(* CODESYS project ChiefMaster.project

Project tree, tasks and I/O mapping:
  Device : HY-TTC 580, TTControl, order no. n/a, version 1.7.1.0
    application Application
      libraries: Standard, * (System); lib500_can2, 0.2.0.5 (TTControl); lib500, 1.7.1.0 (TTControl); lib500_types, 1.7.1.0 (TTControl); lib500_syscom, 1.7.1.0 (TTControl)
      task MainTask (cyclic, interval t#10ms, priority 2, watchdog t#30ms x 1) calls PLC_PRG
      program PLC_PRG [ST]
      global variables GVL
      function block Receive [ST]
      function block Transmit [ST]
      function block Chart [ST]
      global variables GVL_CONSTS
      global variables GVL_VARS
      function block PLC_CODER_TIMER [ST]
      function rt_floorf [ST]
      function block Lib_InputProcessing_state [ST]
      function rt_floord [ST]
      function block Chart1 [ST]
      function block Chart1_l [ST]
      function block Chart_ContactorFB_State_Batt1 [ST]
      function block Chart_lg [ST]
      function block ChiefMaster [ST]
      function block Chart_REQ_IMD_ON_BB1 [ST]
      function block Chart_REQ_IMD_ON_BB2 [ST]
      function block Chart_REQ_IMD_ON_BB3 [ST]
      function block Chart_WeldingDetection [ST]
      function block Chart_j [ST]
      function block VoltageDetermination [ST]
      function PLC_BOOL_TO_LREAL [ST]
      function block InsulationMonitoringReq [ST]
      function block Chart_ek [ST]
      function block Chart_ls [ST]
      function block fcn_EmergencyButtonState [ST]
      function block Chart_REQ_HV_ON_Batt1 [ST]
      function block BattChargeFcn [ST]
      function block Chart_PrechargeStatus [ST]
      function block Chart_REQ_MAIN_MINUS [ST]
      function block SafeToCloseHV [ST]
      function block HVIL_NOK [ST]
      function block Chart_SetDominantSwitch [ST]
      function block Chart_ContactorFB_State_Batt2 [ST]
      function block Chart_ContactorFB_State_Batt3 [ST]
      function block CMState [ST]
      function block EmergencySD [ST]
      function block IMD_SD [ST]
      function block SDError [ST]
      function block Chart_Hysteresis_LowActive [ST]
      function block BDU_Error [ST]
      function block ChartBatt1 [ST]
      function block Chartbatt2 [ST]
      function block ChartBatt3 [ST]
      function block Input_Delay [ST]
      function block Chart_REQ_HV_ON_Batt2 [ST]
      function block Chart_REQ_HV_ON_Batt3 [ST]
      function block REQ_HV_ON_Batt [ST]
      function block Chart_Hysteresis_HighActive [ST]
      function block HVIL_Input_Delay [ST]
      function block IMDOK_Input_Delay [ST]
      function block EMSRET [ST]
      function block EMSRET_Power [ST]
      function block Chart_jj [ST]
      function block Chart_m [ST]
      function block IMD_OK [ST]
      function IMD_Error [ST]
    CANs : CANs, TTControl, order no. n/a, version 1.7.1.0
      CAN0 : CAN0, TTControl, order no. n/a, version 1.7.1.0
      CAN1 : CAN1, TTControl, order no. n/a, version 1.7.1.0
      CAN2 : CAN2, TTControl, order no. n/a, version 1.7.1.0
          settings: Baudrate = 250
      CAN3 : CAN3, TTControl, order no. n/a, version 1.7.1.0
      CAN4 : CAN4, TTControl, order no. n/a, version 1.7.1.0
          settings: Baudrate = 250
      CAN5 : CAN5, TTControl, order no. n/a, version 1.7.1.0
          settings: Baudrate = 250
      CAN6 : CAN6, TTControl, order no. n/a, version 1.7.1.0
    System : System, TTControl, order no. n/a, version 1.7.1.0
        output Application.GVL.gPowerStage : BYTE  // mode
        output Application.GVL.gSafetySwitch0 : BYTE  // mode
        output Application.GVL.gSafetySwitch1 : BYTE  // mode
        output Application.GVL.gSafetySwitch2 : BYTE  // mode
        output Application.GVL.gSensorSupply0 : BYTE  // mode
        output Application.GVL.gSensorSupply1 : BYTE  // mode
        output Application.GVL.gSensorSupply2 : BYTE  // mode
        output TTC_Sleep : BIT  // shutdown
        input  VBat_mV : DWORD  // UBAT.value
        input  KL15_mV : DWORD  // Terminal_15.value
        input  WakeUp_mV : DWORD  // WakeUp.value
        input  WakeUp : BYTE  // WakeUp.state
        unmapped channels: error, error, error, error, error, error, error, error, enable_error_group_0, enable_error_group_1, enable_error_group_2, diag_status, safe_state, error, driver_init_error, UBAT, Terminal_15, WakeUp, Temperature, SSW0, SSW1, SSW2, SSUP0, SSUP1, SSUP2, status, write, boot_error, trigger_error, Powerstage, SSW0, SSW1, SSW2, SSUP0, SSUP1, SSUP2, Terminal_15, WakeUp, ExtShutOff0, ExtShutOff1,
          ExtShutOff2
      Analog_Inputs_2Mode_10V : AIN_2Mode_10V, TTControl, order no. n/a, version 1.7.1.0
        Pin 107
          HVIL_BDU : IoDrvADC2Mode10, TTControl, order no. n/a, version 1.7.1.0
              input  AI_HVIL_BDU_P107 : DWORD  // status.value
              unmapped channels: status, reset_trigger, reset_count, reset_error
        Pin 131
          EmergencyButton_NC : IoDrvADC2Mode10, TTControl, order no. n/a, version 1.7.1.0
              input  AI_EmergencyButton_NC_P131 : DWORD  // status.value
              unmapped channels: status, reset_trigger, reset_count, reset_error
        Pin 108
          HVIL_Components : IoDrvADC2Mode10, TTControl, order no. n/a, version 1.7.1.0
              input  AI_HVIL_Components_P108 : DWORD  // status.value
              unmapped channels: status, reset_trigger, reset_count, reset_error
        Pin 132
          ResetButton_NO : IoDrvDILim, TTControl, order no. n/a, version 1.7.1.0
              input  DI_ResetButton_NO_P132 : BIT  // status.pin_value
              unmapped channels: status
        Pin 109
          HVIL_Battery : IoDrvADC2Mode10, TTControl, order no. n/a, version 1.7.1.0
              input  AI_HVIL_Battery_P109 : DWORD  // status.value
              unmapped channels: status, reset_trigger, reset_count, reset_error
        Pin 133
          Proximity_BB1 : IoDrvDILim, TTControl, order no. n/a, version 1.7.1.0
              input  DI_Proximity_BB1_P133 : BIT  // status.pin_value
              unmapped channels: status
        Pin 110
          HVIL_Overrule : IoDrvDILim, TTControl, order no. n/a, version 1.7.1.0
              input  DI_HVIL_Overrule_P110 : BIT  // status.pin_value
              unmapped channels: status
        Pin 134
          Proximity_BB2 : IoDrvDILim, TTControl, order no. n/a, version 1.7.1.0
              input  DI_Proximity_BB2_P134 : BIT  // status.pin_value
              unmapped channels: status
      Analog_Inputs_2Mode_32V : AIN_2Mode_32V, TTControl, order no. n/a, version 1.7.1.0
        Pin 111
          <Empty>
        Pin 135
          Proximity_BB3 : IoDrvDILim, TTControl, order no. n/a, version 1.7.1.0
              input  DI_Proximity_BB3_P135 : BIT  // status.pin_value
              unmapped channels: status
        Pin 112
          IMD_FB_BB1 : IoDrvDILim, TTControl, order no. n/a, version 1.7.1.0
              input  DI_IMD_FB_BB1_P112 : BIT  // status.pin_value
              unmapped channels: status
        Pin 136
          <Empty>
        Pin 113
          IMD_FB_BB2 : IoDrvDILim, TTControl, order no. n/a, version 1.7.1.0
              input  DI_IMD_FB_BB2_P113 : BIT  // status.pin_value
              unmapped channels: status
        Pin 137
          <Empty>
        Pin 114
          IMD_FB_BB3 : IoDrvDILim, TTControl, order no. n/a, version 1.7.1.0
              input  DI_IMD_FB_BB3_P114 : BIT  // status.pin_value
              unmapped channels: status
        Pin 138
          <Empty>
      Analog_Inputs_3Mode : AIN_3Mode, TTControl, order no. n/a, version 1.7.1.0
        Pin 103
          <Empty>
        Pin 127
          <Empty>
        Pin 104
          <Empty>
        Pin 128
          <Empty>
        Pin 105
          <Empty>
        Pin 129
          <Empty>
        Pin 106
          <Empty>
        Pin 130
          <Empty>
      Digital_Outputs_HS : HSDOUT, TTControl, order no. n/a, version 1.7.1.0
        Pin 149
          KL15_BB1 : IoDrvDOSafety, TTControl, order no. n/a, version 1.7.1.0
              output DO_KL15_BB1_P149 : BIT  // output
              unmapped channels: error_code, reset_trigger, reset_count, reset_error, current, voltage_feedback
        Pin 173
          IMD_BB1 : IoDrvDOSafety, TTControl, order no. n/a, version 1.7.1.0
              output DO_IMD_BB1_P173 : BIT  // output
              unmapped channels: error_code, reset_trigger, reset_count, reset_error, current, voltage_feedback
        Pin 152
          KL15_BB2 : IoDrvDOSafety, TTControl, order no. n/a, version 1.7.1.0
              output DO_KL15_BB2_P152 : BIT  // output
              unmapped channels: error_code, reset_trigger, reset_count, reset_error, current, voltage_feedback
        Pin 176
          IMD_BB2 : IoDrvDOSafety, TTControl, order no. n/a, version 1.7.1.0
              output DO_IMD_BB2_P176 : BIT  // output
              unmapped channels: error_code, reset_trigger, reset_count, reset_error, current, voltage_feedback
        Pin 155
          KL15_BB3 : IoDrvDOSafety, TTControl, order no. n/a, version 1.7.1.0
              output DO_KL15_BB3_P155 : BIT  // output
              unmapped channels: error_code, reset_trigger, reset_count, reset_error, current, voltage_feedback
        Pin 179
          IMD_BB3 : IoDrvDOSafety, TTControl, order no. n/a, version 1.7.1.0
              output DO_IMD_BB3_P179 : BIT  // output
              unmapped channels: error_code, reset_trigger, reset_count, reset_error, current, voltage_feedback
        Pin 158
          <Empty>
        Pin 182
          <Empty>
      Digital_Outputs_LS : LSDOUT, TTControl, order no. n/a, version 1.7.1.0
        Pin 251
          Request_Main_Precharge : IoDrvDO, TTControl, order no. n/a, version 1.7.1.0
              output DO_Request_Main_Precharge_P251 : BIT  // output
              unmapped channels: error_code, reset_trigger, reset_count, reset_error, current
        Pin 238
          Request_Main_Plus : IoDrvDO, TTControl, order no. n/a, version 1.7.1.0
              output DO_Request_Main_Plus_P238 : BIT  // output
              unmapped channels: error_code, reset_trigger, reset_count, reset_error, current
        Pin 252
          <Empty>
        Pin 239
          Request_Main_Minus : IoDrvDO, TTControl, order no. n/a, version 1.7.1.0
              output DO_Request_Main_Minus_P239 : BIT  // output
              unmapped channels: error_code, reset_trigger, reset_count, reset_error, current
        Pin 253
          <Empty>
        Pin 240
          Request_DC_Plus : IoDrvDO, TTControl, order no. n/a, version 1.7.1.0
              output DO_Request_DC_Plus_P240 : BIT  // output
              unmapped channels: error_code, reset_trigger, reset_count, reset_error, current
        Pin 254
          <Empty>
        Pin 241
          Request_DC_Minus : IoDrvDO, TTControl, order no. n/a, version 1.7.1.0
              output DO_Request_DC_Minus_P241 : BIT  // output
              unmapped channels: error_code, reset_trigger, reset_count, reset_error, current
      PVG_Outputs : PVG, TTControl, order no. n/a, version 1.7.1.0
        Pin 161
          HVIL_Supply : IoDrvDODiag, TTControl, order no. n/a, version 1.7.1.0
              settings: diagnostic = FALSE
              output DO_HVIL_Supply_P161 : BIT  // output
              unmapped channels: error_code, reset_trigger, reset_count, reset_error, current, voltage_feedback
        Pin 185
          ResetButton_LED : IoDrvDODiag, TTControl, order no. n/a, version 1.7.1.0
              settings: diagnostic = FALSE
              output DO_REsetButton_LED_P185 : BIT  // output
              unmapped channels: error_code, reset_trigger, reset_count, reset_error, current, voltage_feedback
        Pin 188
          CabinAlarm : IoDrvDODiag, TTControl, order no. n/a, version 1.7.1.0
              settings: diagnostic = FALSE
              output DO_CabinAlarm_P188 : BIT  // output
              unmapped channels: error_code, reset_trigger, reset_count, reset_error, current, voltage_feedback
        Pin 164
          <Empty>
        Pin 191
          <Empty>
        Pin 167
          <Empty>
        Pin 194
          <Empty>
        Pin 170
          <Empty>
      PWM_Outputs : PWM, TTControl, order no. n/a, version 1.7.1.0
        Safety_switch_0 : PWM_SSW0, TTControl, order no. n/a, version 1.7.1.0
          Pin 153
            <Empty>
          Pin 177
            HeaterPump : IoDrvDO, TTControl, order no. n/a, version 1.7.1.0
                output DO_HeaterPump_Active_Pin177 : BIT  // output
                unmapped channels: error_code, reset_trigger, reset_count, reset_error, current
          Pin 156
            <Empty>
          Pin 180
            Alternator_ouput : IoDrvDO, TTControl, order no. n/a, version 1.7.1.0
                output DO_AlternatorOutput_Pin180 : BIT  // output
                unmapped channels: error_code, reset_trigger, reset_count, reset_error, current
          Pin 159
            <Empty>
          Pin 183
            CoolingSystemPump : IoDrvDO, TTControl, order no. n/a, version 1.7.1.0
                output DO_CoolingSystemPump_Pin183 : BIT  // output
                unmapped channels: error_code, reset_trigger, reset_count, reset_error, current
          Pin 186
            CoolingSystemFan : IoDrvDO, TTControl, order no. n/a, version 1.7.1.0
                output DO_CoolingSystemFan_Pin186 : BIT  // output
                unmapped channels: error_code, reset_trigger, reset_count, reset_error, current
          Pin 162
            <Empty>
          Pin 189
            HydraulicFan : IoDrvDO, TTControl, order no. n/a, version 1.7.1.0
                output DO_HydraulicFan_Pin189 : BIT  // output
                unmapped channels: error_code, reset_trigger, reset_count, reset_error, current
          Pin 165
            <Empty>
          Pin 192
            BMS_KL15 : IoDrvDO, TTControl, order no. n/a, version 1.7.1.0
                output DO_BMSKL15_Pin192 : BIT  // output
                unmapped channels: error_code, reset_trigger, reset_count, reset_error, current
          Pin 168
            <Empty>
          Pin 195
            <Empty>
          Pin 171
            <Empty>
        Safety_switch_1 : PWM_SSW1, TTControl, order no. n/a, version 1.7.1.0
          Pin 154
            <Empty>
          Pin 178
            <Empty>
          Pin 157
            <Empty>
          Pin 181
            <Empty>
          Pin 160
            <Empty>
          Pin 184
            <Empty>
          Pin 187
            <Empty>
          Pin 163
            <Empty>
          Pin 190
            <Empty>
          Pin 166
            <Empty>
          Pin 193
            <Empty>
          Pin 169
            <Empty>
          Pin 196
            <Empty>
          Pin 172
            <Empty>
        Safety_switch_2 : PWM_SSW2, TTControl, order no. n/a, version 1.7.1.0
          Pin 101
            EMSRET_BDU1 : IoDrvDO, TTControl, order no. n/a, version 1.7.1.0
                output DO_EMSRET_BDU1 : BIT  // output
                unmapped channels: error_code, reset_trigger, reset_count, reset_error, current
          Pin 125
            EMSRET_BDU2 : IoDrvDO, TTControl, order no. n/a, version 1.7.1.0
                output DO_EMSRET_BDU2 : BIT  // output
                unmapped channels: error_code, reset_trigger, reset_count, reset_error, current
          Pin 150
            EMSRET_BB2_1 : IoDrvDO, TTControl, order no. n/a, version 1.7.1.0
                output DO_EMSRET_BB2_1 : BIT  // output
                unmapped channels: error_code, reset_trigger, reset_count, reset_error, current
          Pin 174
            EMSRET_BB2_2 : IoDrvDO, TTControl, order no. n/a, version 1.7.1.0
                output DO_EMSRET_BB2_2 : BIT  // output
                unmapped channels: error_code, reset_trigger, reset_count, reset_error, current
          Pin 102
            EMSRET_BB1_1 : IoDrvDO, TTControl, order no. n/a, version 1.7.1.0
                output DO_EMSRET_BB1_1 : BIT  // output
                unmapped channels: error_code, reset_trigger, reset_count, reset_error, current
          Pin 126
            EMSRET_BB1_2 : IoDrvDO, TTControl, order no. n/a, version 1.7.1.0
                output DO_EMSRET_BB1_2 : BIT  // output
                unmapped channels: error_code, reset_trigger, reset_count, reset_error, current
          Pin 151
            EMSRET_BB3_1 : IoDrvDO, TTControl, order no. n/a, version 1.7.1.0
                output DO_EMSRET_BB3_1 : BIT  // output
                unmapped channels: error_code, reset_trigger, reset_count, reset_error, current
          Pin 175
            EMSRET_BB3_2 : IoDrvDO, TTControl, order no. n/a, version 1.7.1.0
                output DO_EMSRET_BB3_2 : BIT  // output
                unmapped channels: error_code, reset_trigger, reset_count, reset_error, current
      Timer_Inputs_Cur : TIN_Cur, TTControl, order no. n/a, version 1.7.1.0
        Pin 115
          Main_Plus_FB : IoDrvADC, TTControl, order no. n/a, version 1.7.1.0
              input  AI_Main_Plus_FB_P115 : DWORD  // status.value
              unmapped channels: status
        Pin 139
          <Empty>
        Pin 116
          Main_Minus_FB : IoDrvADC, TTControl, order no. n/a, version 1.7.1.0
              input  AI_Main_Minus_FB_P116 : DWORD  // status.value
              unmapped channels: status
        Pin 140
          <Empty>
        Pin 117
          <Empty>
        Pin 141
          <Empty>
      Timer_Inputs : TIN, TTControl, order no. n/a, version 1.7.1.0
        Pin 122
          DC_Plus_FB : IoDrvADC, TTControl, order no. n/a, version 1.7.1.0
              input  AI_DC_Plus_FB_P122 : DWORD  // status.value
              unmapped channels: status
        Pin 146
          <Empty>
        Pin 123
          DC_Minus_FB : IoDrvADC, TTControl, order no. n/a, version 1.7.1.0
              input  AI_DC_Minus_FB_P123 : DWORD  // status.value
              unmapped channels: status
        Pin 147
          <Empty>
        Pin 124
          <Empty>
        Pin 148
          <Empty>
*)

// Device/Application/GVL
 {attribute 'qualified_only'}
VAR_GLOBAL
	(*System*)
	gPowerStage    : lib500_types.IO_POWER_STATE := lib500_types.IO_POWER_STATE.IO_POWER_OFF;	(* Powerstage status variable *)
	gSafetySwitch0 : lib500_types.IO_POWER_STATE := lib500_types.IO_POWER_STATE.IO_POWER_OFF;   (* Safey Switch 0 status variable *)
	gSafetySwitch1 : lib500_types.IO_POWER_STATE := lib500_types.IO_POWER_STATE.IO_POWER_OFF;   (* Safey Switch 1 status variable *)
	gSafetySwitch2 : lib500_types.IO_POWER_STATE := lib500_types.IO_POWER_STATE.IO_POWER_OFF;   (* Safey Switch 2 status variable *)
	gSensorSupply0 : lib500_types.IO_POWER_STATE := lib500_types.IO_POWER_STATE.IO_POWER_OFF;   (* Sensor Supply status variable *)
	gSensorSupply1 : lib500_types.IO_POWER_STATE := lib500_types.IO_POWER_STATE.IO_POWER_OFF;   (* Sensor Supply status variable *)
	gSensorSupply2 : lib500_types.IO_POWER_STATE := lib500_types.IO_POWER_STATE.IO_POWER_OFF;   (* Sensor Supply status variable *)
	G_tonCMSleep_timer:TON;
	G_CMSleep: BOOL;
	
(*CAN*)
	gCan0: tCan;
	gCan1: tCan;
	gCan2: tCan;
	gCan3: tCan;
	gCan4: tCan;
	gCan5: tCan;

	(*Recieve*)
	
(*Actia*)
(*Box 1*)
	C_Actia_BB1_MyStatus: ARRAY [0..7] OF BYTE;
	C_Actia_BB1_MyStatus_Timeout: BOOL;
	C_Actia_BB1_Error: ARRAY [0..7] OF BYTE;
	C_Actia_BB1_Error_Timeout: BOOL;
	C_Actia_BB1_ADS_8: ARRAY [0..7] OF BYTE;
	C_Actia_BB1_ADS_8_Timeout: BOOL;
	C_Actia_BB1_ADS_0: ARRAY [0..7] OF BYTE;
	C_Actia_BB1_ADS_0_Timeout: BOOL;
	C_Actia_BB1_ADS_1: ARRAY [0..7] OF BYTE;
	C_Actia_BB1_ADS_1_Timeout: BOOL;
	C_Actia_BB1_ADS_3: ARRAY [0..7] OF BYTE;
	C_Actia_BB1_ADS_3_Timeout: BOOL;
(*Box 2*)
	C_Actia_BB2_MyStatus: ARRAY [0..7] OF BYTE;
	C_Actia_BB2_MyStatus_Timeout: BOOL;
	C_Actia_BB2_Error: ARRAY [0..7] OF BYTE;
	C_Actia_BB2_Error_Timeout: BOOL;
	C_Actia_BB2_ADS_8: ARRAY [0..7] OF BYTE;
	C_Actia_BB2_ADS_8_Timeout: BOOL;
	C_Actia_BB2_ADS_0: ARRAY [0..7] OF BYTE;
	C_Actia_BB2_ADS_0_Timeout: BOOL;
	C_Actia_BB2_ADS_1: ARRAY [0..7] OF BYTE;
	C_Actia_BB2_ADS_1_Timeout: BOOL;
	C_Actia_BB2_ADS_3: ARRAY [0..7] OF BYTE;
	C_Actia_BB2_ADS_3_Timeout: BOOL;
(*Box 3*)	
	C_Actia_BB3_MyStatus: ARRAY [0..7] OF BYTE;
	C_Actia_BB3_MyStatus_Timeout: BOOL;
	C_Actia_BB3_Error: ARRAY [0..7] OF BYTE;
	C_Actia_BB3_Error_Timeout: BOOL;
	C_Actia_BB3_ADS_8: ARRAY [0..7] OF BYTE;
	C_Actia_BB3_ADS_8_Timeout: BOOL;
	C_Actia_BB3_ADS_0: ARRAY [0..7] OF BYTE;
	C_Actia_BB3_ADS_0_Timeout: BOOL;
	C_Actia_BB3_ADS_1: ARRAY [0..7] OF BYTE;
	C_Actia_BB3_ADS_1_Timeout: BOOL;
	C_Actia_BB3_ADS_3: ARRAY [0..7] OF BYTE;
	C_Actia_BB3_ADS_3_Timeout: BOOL;
	
(*LiBa*)
(*Box 1*)
	C_LB_Batt1_CellVoltage01: ARRAY[0..7] OF BYTE;
	C_LB_Batt1_CellVoltage01_Timeout: BOOL;
	C_LB_Batt1_CellVoltage02: ARRAY[0..7] OF BYTE;
	C_LB_Batt1_CellVoltage02_Timeout: BOOL;
	C_LB_Batt1_CellTemperature: ARRAY[0..7] OF BYTE;
	C_LB_Batt1_CellTemperature_Timeout: BOOL;
	C_LB_Batt1_InsulationMonitor: ARRAY[0..7] OF BYTE;
	C_LB_Batt1_InsulationMonitor_Timeout: BOOL;
	C_LB_Batt1_Status01: ARRAY[0..7] OF BYTE;
	C_LB_Batt1_Status01_Timeout: BOOL;
	C_LB_Batt1_Status02: ARRAY[0..7] OF BYTE;
	C_LB_Batt1_Status02_Timeout: BOOL;
	C_LB_Batt1_Status03: ARRAY[0..7] OF BYTE;
	C_LB_Batt1_Status03_Timeout: BOOL;

(*Box 2*)
	C_LB_Batt2_CellVoltage01: ARRAY[0..7] OF BYTE;
	C_LB_Batt2_CellVoltage01_Timeout: BOOL;
	C_LB_Batt2_CellVoltage02: ARRAY[0..7] OF BYTE;
	C_LB_Batt2_CellVoltage02_Timeout: BOOL;
	C_LB_Batt2_CellTemperature: ARRAY[0..7] OF BYTE;
	C_LB_Batt2_CellTemperature_Timeout: BOOL;
	C_LB_Batt2_InsulationMonitor: ARRAY[0..7] OF BYTE;
	C_LB_Batt2_InsulationMonitor_Timeout: BOOL;
	C_LB_Batt2_Status01: ARRAY[0..7] OF BYTE;
	C_LB_Batt2_Status01_Timeout: BOOL;
	C_LB_Batt2_Status02: ARRAY[0..7] OF BYTE;
	C_LB_Batt2_Status02_Timeout: BOOL;
	C_LB_Batt2_Status03: ARRAY[0..7] OF BYTE;
	C_LB_Batt2_Status03_Timeout: BOOL;

(*Box 3*)
	C_LB_Batt3_CellVoltage01: ARRAY[0..7] OF BYTE;
	C_LB_Batt3_CellVoltage01_Timeout: BOOL;
	C_LB_Batt3_CellVoltage02: ARRAY[0..7] OF BYTE;
	C_LB_Batt3_CellVoltage02_Timeout: BOOL;
	C_LB_Batt3_CellTemperature: ARRAY[0..7] OF BYTE;
	C_LB_Batt3_CellTemperature_Timeout: BOOL;
	C_LB_Batt3_InsulationMonitor: ARRAY[0..7] OF BYTE;
	C_LB_Batt3_InsulationMonitor_Timeout: BOOL;
	C_LB_Batt3_Status01: ARRAY[0..7] OF BYTE;
	C_LB_Batt3_Status01_Timeout: BOOL;
	C_LB_Batt3_Status02: ARRAY[0..7] OF BYTE;
	C_LB_Batt3_Status02_Timeout: BOOL;
	C_LB_Batt3_Status03: ARRAY[0..7] OF BYTE;
	C_LB_Batt3_Status03_Timeout: BOOL;
	
(*UDC*)	
	C_UDC_Msg1: ARRAY[0..7] OF BYTE;
	C_UDC_Msg1_Timeout: BOOL;
	
(*Transmit*)
(*Actia*)
	C_Actia_Control_Batt1 : ARRAY[0..7] OF BYTE;
	C_Actia_Control_Batt2 : ARRAY[0..7] OF BYTE;
	C_Actia_Control_Batt3 : ARRAY[0..7] OF BYTE;
(*LiBa*)
	C_LiBa_OperationRequest_Batt1: ARRAY[0..7] OF BYTE;
	C_LiBa_OperationRequest_Batt2: ARRAY[0..7] OF BYTE;
	C_LiBa_OperationRequest_Batt3: ARRAY[0..7] OF BYTE;
(*Chief Master*)
	C_Chief_Master_Msg1 : ARRAY[0..7] OF BYTE;
	C_Chief_Master_Msg2 : ARRAY[0..7] OF BYTE;
	C_Chief_Master_Msg3 : ARRAY[0..7] OF BYTE;
	C_Chief_Master_Msg4 : ARRAY[0..7] OF BYTE;
	C_Chief_Master_Msg5 : ARRAY[0..7] OF BYTE;
	C_Chief_Master_Msg6 : ARRAY[0..7] OF BYTE;
	C_Chief_Master_Msg7 : ARRAY[0..7] OF BYTE;
	C_Chief_Master_Msg8 : ARRAY[0..7] OF BYTE;
	C_Chief_Master_Msg9 : ARRAY[0..7] OF BYTE;
	C_Chief_Master_Msg10: ARRAY[0..7] OF BYTE;
	C_Chief_Master_Msg11: ARRAY[0..7] OF BYTE;
	C_Chief_Master_Msg12: ARRAY[0..7] OF BYTE;
	C_Chief_Master_Msg13: ARRAY[0..7] OF BYTE;
	C_Chief_Master_Msg14: ARRAY[0..7] OF BYTE;
	C_Chief_Master_Msg15: ARRAY[0..7] OF BYTE;

END_VAR

// Device/Application/GVL_CONSTS
VAR_GLOBAL CONSTANT
	ChiefMaster_IN_Default_e2: USINT := 1;
	ChiefMaster_IN_PrechargeDisable: USINT := 2;
	ChiefMaster_IN_PrechargeEnable: USINT := 3;
	ChiefMaster_IN_NO_ACTIVE_CHILD_f: USINT := 0;
	ChiefMaster_IN_Error_p: USINT := 2;
	ChiefMaster_IN_closed: USINT := 3;
	ChiefMaster_IN_hold_a: USINT := 4;
	ChiefMaster_IN_hold1: USINT := 5;
	ChiefMaster_IN_open: USINT := 6;
	ChiefMaster_IN_Default1: USINT := 2;
	ChiefMaster_IN_Actual_o: USINT := 1;
	ChiefMaster_IN_Default_i2: USINT := 2;
	ChiefMaster_IN_hold_oa: USINT := 3;
	ChiefMaster_IN_BuzzerOFF: USINT := 1;
	ChiefMaster_IN_BuzzerON: USINT := 2;
	SS_OUTPUT: SINT := 3;
	SS_INITIALIZE: SINT := 0;
	SS_UPDATE: SINT := 4;
	ChiefMaster_IN_Default: USINT := 1;
	ChiefMaster_IN_PrechargeFail: USINT := 2;
	ChiefMaster_IN_PrechargeSuccess: USINT := 3;
	ChiefMaster_IN_delay1: USINT := 4;
	ChiefMaster_IN_NO_ACTIVE_CHILD: USINT := 0;
	ChiefMaster_IN_Default_a: USINT := 1;
	ChiefMaster_IN_Hold: USINT := 2;
	ChiefMaster_IN_RELMinusClose: USINT := 3;
	ChiefMaster_IN_NO_ACTIVE_CHILD_h: USINT := 0;
	ChiefMaster_IN_Default_b: USINT := 1;
	ChiefMaster_IN_Default3: USINT := 2;
	ChiefMaster_IN_Error: USINT := 3;
	ChiefMaster_IN_ErrorMinus: USINT := 4;
	ChiefMaster_IN_ErrorPlus: USINT := 5;
	ChiefMaster_IN_ErrorVoltage: USINT := 6;
	ChiefMaster_IN_Minus_Close: USINT := 7;
	b_ChiefMaster_IN_Open: USINT := 8;
	ChiefMaster_IN_Open1: USINT := 9;
	ChiefMaster_IN_Plus_Close: USINT := 10;
	ChiefMaster_IN_NO_ACTIVE_CHILD_e: USINT := 0;
	ChiefMaster_IN_Error_l: USINT := 1;
	ChiefMaster_IN_Open_m: USINT := 2;
	b_ChiefMaster_IN_default: USINT := 3;
	b_ChiefMaster_IN_hold: USINT := 4;
	ChiefMaster_IN_NO_ACTIVE_CHILD_m: USINT := 0;
	ChiefMaster_IN_Error_e: USINT := 1;
	ChiefMaster_IN_Open_p: USINT := 2;
	ChiefMaster_IN_default_h: USINT := 3;
	ChiefMaster_IN_hold_o: USINT := 4;
	ChiefMaster_IN_NO_ACTIVE_CHILD_hs: USINT := 0;
	ChiefMaster_IN_Error_c: USINT := 1;
	ChiefMaster_IN_Open_n: USINT := 2;
	ChiefMaster_IN_default_n: USINT := 3;
	ChiefMaster_IN_hold_h: USINT := 4;
	ChiefMaster_IN_NO_ACTIVE_CHILD_i: USINT := 0;
	ChiefMaster_IN_CONTACTOR_OFF: USINT := 1;
	ChiefMaster_IN_CONTACTOR_ON: USINT := 2;
	b_ChiefMaster_IN_Default_h: USINT := 3;
	ChiefMaster_IN_hold_hp: USINT := 4;
	ChiefMaster_IN_NO_ACTIVE_CHILD_d: USINT := 0;
	ChiefMaster_IN_CONTACTOR_OFF_p: USINT := 1;
	ChiefMaster_IN_CONTACTOR_ON_o: USINT := 2;
	b_ChiefMaster_IN_Default_n: USINT := 3;
	ChiefMaster_IN_hold_i: USINT := 4;
	ChiefMaster_IN_NO_ACTIVE_CHILD_iv: USINT := 0;
	ChiefMaster_IN_CONTACTOR_OFF_f: USINT := 1;
	ChiefMaster_IN_CONTACTOR_ON_b: USINT := 2;
	ChiefMaster_IN_Default_f: USINT := 3;
	ChiefMaster_IN_hold_k: USINT := 4;
	ChiefMaster_IN_NO_ACTIVE_CHILD_k: USINT := 0;
	ChiefMaster_IN_Actual: USINT := 1;
	ChiefMaster_IN_Default_e: USINT := 2;
	b_ChiefMaster_IN_Hold_h: USINT := 3;
	ChiefMaster_IN_NO_ACTIVE_CHILD_j: USINT := 0;
	ChiefMaster_IN_CHARGE: USINT := 1;
	ChiefMaster_IN_DRIVE: USINT := 2;
	ChiefMaster_IN_Default_fx: USINT := 3;
	ChiefMaster_IN_IMD_OFF: USINT := 2;
	ChiefMaster_IN_IMD_ON: USINT := 3;
	ChiefMaster_IN_DRIVE_d: USINT := 1;
	ChiefMaster_IN_NO_ACTIVE_CHILD_a: USINT := 0;
	ChiefMaster_IN_CHARGE_c: USINT := 1;
	ChiefMaster_IN_DRIVE_k: USINT := 2;
	ChiefMaster_IN_Default_d: USINT := 3;
	ChiefMaster_IN_IMD_OFF_m: USINT := 2;
	ChiefMaster_IN_IMD_ON_b: USINT := 3;
	ChiefMaster_IN_DRIVE_ke: USINT := 1;
	ChiefMaster_IN_NO_ACTIVE_CHILD_jz: USINT := 0;
	ChiefMaster_IN_CHARGE_a: USINT := 1;
	ChiefMaster_IN_DRIVE_e: USINT := 2;
	ChiefMaster_IN_Default_j: USINT := 3;
	ChiefMaster_IN_IMD_OFF_a: USINT := 2;
	ChiefMaster_IN_IMD_ON_k: USINT := 3;
	ChiefMaster_IN_DRIVE_e3: USINT := 1;
	ChiefMaster_IN_NO_ACTIVE_CHILD_g: USINT := 0;
	ChiefMaster_IN_Default_o: USINT := 1;
	ChiefMaster_IN_hold_g: USINT := 2;
	ChiefMaster_IN_NO_ACTIVE_CHILD_mp: USINT := 0;
	ChiefMaster_IN_Default_m: USINT := 1;
	ChiefMaster_IN_Delay: USINT := 2;
	b_ChiefMaster_IN_Delay1: USINT := 3;
	ChiefMaster_IN_NO_ACTIVE_CHILD_a4: USINT := 0;
	ChiefMaster_IN_Default_dh: USINT := 1;
	ChiefMaster_IN_Delay_j: USINT := 2;
	ChiefMaster_IN_pulse: USINT := 3;
	ChiefMaster_IN_NO_ACTIVE_CHILD_kt: USINT := 0;
	ChiefMaster_IN_Default_e0: USINT := 1;
	ChiefMaster_IN_Delay_i: USINT := 2;
	ChiefMaster_IN_KL15_reset: USINT := 3;
	ChiefMaster_IN_hold_hw: USINT := 4;
	ChiefMaster_IN_pulse_i: USINT := 5;
	ChiefMaster_IN_NO_ACTIVE_CHILD_a0: USINT := 0;
	ChiefMaster_IN_Default_g: USINT := 1;
	ChiefMaster_IN_Delay_m: USINT := 2;
	ChiefMaster_IN_Delay1_h: USINT := 3;
	ChiefMaster_IN_NO_ACTIVE_CHILD_a1: USINT := 0;
	ChiefMaster_IN_Error_o: USINT := 1;
	ChiefMaster_IN_OFF: USINT := 2;
	ChiefMaster_IN_ON: USINT := 3;
	ChiefMaster_IN_Sleep: USINT := 4;
	ChiefMaster_IN_BDURelayClose: USINT := 1;
	ChiefMaster_IN_BDURelayClose_Req: USINT := 2;
	ChiefMaster_IN_BattRelayClose: USINT := 3;
	ChiefMaster_IN_BattRelayClose_Req: USINT := 4;
	ChiefMaster_IN_ISOMonitor_OK: USINT := 5;
	ChiefMaster_IN_ISOMonitor_check: USINT := 6;
	ChiefMaster_IN_KL15ON: USINT := 7;
	ChiefMaster_IN_BDURelayOpen: USINT := 1;
	ChiefMaster_IN_BDURelayOpen_Req: USINT := 2;
	ChiefMaster_IN_BattRelayOpen: USINT := 3;
	ChiefMaster_IN_BattRelayOpen_Req: USINT := 4;
	ChiefMaster_IN_ISOMonitorOFF: USINT := 5;
	ChiefMaster_IN_KL15OFF: USINT := 6;
	ChiefMaster_IN_NO_ACTIVE_CHILD_ktp: USINT := 0;
	ChiefMaster_IN_Batt1: USINT := 1;
	ChiefMaster_IN_Batt2: USINT := 2;
	ChiefMaster_IN_Batt3: USINT := 3;
	ChiefMaster_IN_Default_b0: USINT := 4;
	ChiefMaster_IN_RampDown: USINT := 5;
	ChiefMaster_IN_Stop: USINT := 6;
	ChiefMaster_IN_NO_ACTIVE_CHILD_c: USINT := 0;
	ChiefMaster_IN_Delay_b: USINT := 1;
	ChiefMaster_IN_OFF_i: USINT := 2;
	ChiefMaster_IN_ON_g: USINT := 3;
	ChiefMaster_IN_ShutOff: USINT := 4;
	ChiefMaster_IN_NO_ACTIVE_CHILD_jr: USINT := 0;
	ChiefMaster_IN_Initial_state: USINT := 1;
	ChiefMaster_IN_Reset_state: USINT := 2;
	ChiefMaster_IN_state1: USINT := 3;
	ChiefMaster_IN_state2: USINT := 4;
	ChiefMaster_IN_NO_ACTIVE_CHILD_b: USINT := 0;
	ChiefMaster_IN_Initial_state_g: USINT := 1;
	ChiefMaster_IN_Reset_state_b: USINT := 2;
	ChiefMaster_IN_state1_o: USINT := 3;
	ChiefMaster_IN_state2_e: USINT := 4;
	ChiefMaster_IN_NO_ACTIVE_CHILD_cn: USINT := 0;
	ChiefMaster_IN_After_delay: USINT := 1;
	ChiefMaster_IN_Delay_a: USINT := 2;
	ChiefMaster_IN_Initial: USINT := 3;
	ChiefMaster_IN_NO_ACTIVE_CHILD_l: USINT := 0;
	ChiefMaster_IN_Default_jp: USINT := 1;
	ChiefMaster_IN_IsoMonitorCheck: USINT := 2;
	ChiefMaster_IN_IsoMonitorError: USINT := 3;
	ChiefMaster_IN_NO_ACTIVE_CHILD_eq: USINT := 0;
	ChiefMaster_IN_Actual_e: USINT := 1;
	ChiefMaster_IN_Default_h3: USINT := 2;
	ChiefMaster_IN_hold_n: USINT := 3;
	ChiefMaster_IN_NO_ACTIVE_CHILD_ir: USINT := 0;
	ChiefMaster_IN_Default_fd: USINT := 1;
	ChiefMaster_IN_Error_ex: USINT := 2;
	ChiefMaster_IN_NO_ACTIVE_CHILD_cs: USINT := 0;
	ChiefMaster_IN_HighValue: USINT := 1;
	ChiefMaster_IN_LowValue: USINT := 2;
	ChiefMaster_IN_OFF_c: USINT := 3;
	ChiefMaster_IN_NO_ACTIVE_CHILD_p: USINT := 0;
	ChiefMaster_IN_After_delay_c: USINT := 1;
	ChiefMaster_IN_Delay_k: USINT := 2;
	ChiefMaster_IN_Initial_h: USINT := 3;
	ChiefMaster_IN_NO_ACTIVE_CHILD_cr: USINT := 0;
	ChiefMaster_IN_HighValue_a: USINT := 1;
	ChiefMaster_IN_LowValue_n: USINT := 2;
	ChiefMaster_IN_OFF_o: USINT := 3;
	ChiefMaster_IN_NO_ACTIVE_CHILD_i2: USINT := 0;
	ChiefMaster_IN_After_delay_p: USINT := 1;
	ChiefMaster_IN_Initial_k: USINT := 2;
	ChiefMaster_IN_NO_ACTIVE_CHILD_an: USINT := 0;
	SS_DISABLE: SINT := 6;
	ChiefMaster_IN_Actia: USINT := 1;
	ChiefMaster_IN_Default_at: USINT := 2;
	ChiefMaster_IN_LiBa: USINT := 3;
	ChiefMaster_IN_NO_ACTIVE_CHILD_i3: USINT := 0;
	ChiefMaster_IN_Actia_m: USINT := 1;
	ChiefMaster_IN_Default_jw: USINT := 2;
	ChiefMaster_IN_LiBa_h: USINT := 3;
	ChiefMaster_IN_NO_ACTIVE_CHILD_d4: USINT := 0;
	ChiefMaster_IN_Actia_p: USINT := 1;
	ChiefMaster_IN_Default_bc: USINT := 2;
	ChiefMaster_IN_LiBa_d: USINT := 3;
	ChiefMaster_IN_NO_ACTIVE_CHILD_gp: USINT := 0;
	ChiefMaster_IN_After_delay1: USINT := 1;
	ChiefMaster_IN_Initial1: USINT := 2;
	ChiefMaster_IN_NO_ACTIVE_CHILD_jg: USINT := 0;
	ChiefMaster_IN_Default_i: USINT := 1;
	ChiefMaster_IN_Hold_m: USINT := 2;
	ChiefMaster_IN_Hold2: USINT := 3;
	ChiefMaster_IN_Hold3: USINT := 4;
	ChiefMaster_IN_NO_ACTIVE_CHILD_gd: USINT := 0;
	SS_STEP: SINT := 1;
END_VAR

// Device/Application/GVL_VARS
VAR_GLOBAL
	OP_boHVIL_Supply: BOOL := TRUE;
	FL_sHVC_CellBalanceVoltage_mV: REAL := 3500.0;
	VoltageSensorAvailableBB1: BOOL;
	VoltageSensorAvailableBB2: BOOL;
	VoltageSensorAvailableBB3: BOOL;
	NotAvailable_uint16: REAL := 65535.0;
	UnexpectedBattChargingFcn_Available: BOOL := TRUE;
	CurrentReductionConstant_Lvl3: REAL := 0.1;
	NotAvailable_uint8: USINT := 255;
	MainHV_Minus_In_Delay: REAL := 5.0;
	MainHV_StatusDelay: REAL := 5.0;
	DCHV_Minus_In_Delay_ms: REAL := 500.0;
	FL_u8HMI_BuzzerTimer: USINT := 3;
	CurrentReductionConstant_Lvl2: REAL := 0.07;
	CurrentReductionConstant_Lvl1: REAL := 0.05;
	CurrentReductionConstant_Lvl0: REAL := 0.03;
	IT_u8IMD_DelayTime_s: USINT := 20;
	CurrentLB: REAL := -3.0;
	CurrentUB: REAL := 3.0;
	IP_u8HVIL_Delay_ms: USINT := 100;
	IP_u8HW_IN_delay_ms: USINT := 100;
	FL_sInrushCurrent_dividebyzero: REAL := 1.0E-5;
	SafeVoltageToCloseHV_V: REAL := 0.5;
	SafeCurrentToCloseHV_A: REAL := 5.0;
	BattBox1_No: REAL := 1.0;
	BattBox2_No: REAL := 2.0;
	BattBox3_No: REAL := 3.0;
	Voltage_NA_UB: UINT := 65535;
END_VAR

// Device/Application/PLC_PRG
PROGRAM PLC_PRG
VAR
	InitPowerstages:BOOL:= TRUE;
	InitCAN0:BOOL:= TRUE;
	InitCAN1:BOOL:= TRUE;
	InitCAN2:BOOL:= TRUE;
	InitCAN3:BOOL:= TRUE;
	InitCAN4:BOOL:= TRUE;
	InitCAN5:BOOL:= TRUE;
	Receive_Msg: Receive;
	Transmit_Msg: Transmit;
	ChiefMaster: ChiefMaster;
END_VAR

(*PLC Initialization*)
IF (InitPowerstages = TRUE) THEN
	GVL.gPowerStage 	:= lib500_types.IO_POWER_STATE.IO_POWER_ON;		(* Switching on Power Stage *)
	GVL.gSensorSupply0  := lib500_types.IO_POWER_STATE.IO_POWER_ON;		(* Switching on Sensor Supply 0 to get 5V for Potentiometer *)
	GVL.gSensorSupply1  := lib500_types.IO_POWER_STATE.IO_POWER_ON;		(* Switching on Sensor Supply 1 to get 5V for Potentiometer *)
	GVL.gSensorSupply2  := lib500_types.IO_POWER_STATE.IO_POWER_ON_10V;	(* Switching on Sensor Supply 2 to get 10V for Potentiometer *)
    GVL.gSafetySwitch0 	:= lib500_types.IO_POWER_STATE.IO_POWER_ON;     (* Switching on Safety Switch 0 for PWM use *)
	GVL.gSafetySwitch1 	:= lib500_types.IO_POWER_STATE.IO_POWER_ON; 	(* Switching on Safety Switch 1 for PWM use *)
	GVL.gSafetySwitch2 	:= lib500_types.IO_POWER_STATE.IO_POWER_ON; 	(* Switching on Safety Switch 2 for PWM use *)
	InitPowerstages:= FALSE;
END_IF
IF (InitCAN0 = TRUE) THEN
	CanInit(	iEnable			:= TRUE,                        (* Initialiaze CAN *)
				iChannel		:= 0,							(* CAN Channel 0 *)
				iCAN			:= ADR(GVL.gCan0), 				(* Structure for sending / receiving CAN messages *)
				iBaudrate		:= 250,							(* 250 kBit *)
				iCanIdExtended	:= FALSE,						(* Standard CAN Frame *)
				iEcuCycleTime  	:= T#10MS);						(* Cycle time of task calling TX and RX *)
	InitCAN0 := FALSE;											(* Execute this block one time for initialisation *)
END_IF
IF (InitCAN1 = TRUE) THEN
	CanInit(	iEnable			:= TRUE,                        (* Initialiaze CAN *)
				iChannel		:= 1,							(* CAN Channel 1 *)
				iCAN			:= ADR(GVL.gCan1), 				(* Structure for sending / receiving CAN messages *)
				iBaudrate		:= 500,							(* 500 kBit *)
				iCanIdExtended	:= FALSE,						(* Standard CAN Frame *)
				iEcuCycleTime  	:= T#10MS);						(* Cycle time of task calling TX and RX *)
	InitCAN1 := FALSE;											(* Execute this block one time for initialisation *)
END_IF
IF (InitCAN2 = TRUE) THEN 
	CanInit(	iEnable			:= TRUE,                  		(* Initialiaze CAN *)
				iChannel		:= 2,							(* CAN Channel 2 *)
				iCAN			:= ADR(GVL.gCan2), 				(* Structure for sending / receiving CAN messages *)
				iBaudrate       := 500, 					    (* 250 kBit *)
				iCanIdExtended  := FALSE, 						(* Standard CAN Frame *)
				iEcuCycleTime  	:= T#10MS);						(* Cycle time of task calling TX and RX *)
	InitCAN2 := FALSE;											(* Execute this block one time for initialisation *)
END_IF					
IF (InitCAN3 = TRUE) THEN 
	CanInit(	iEnable			:= TRUE,                  		(* Initialiaze CAN *)
				iChannel		:= 3,							(* CAN Channel 3 *)
				iCAN			:= ADR(GVL.gCan3), 				(* Structure for sending / receiving CAN messages *)
				iBaudrate       := 500, 					    (* 250 kBit *)
				iCanIdExtended  := FALSE, 						(* Standard CAN Frame *)
				iEcuCycleTime  	:= T#10MS);						(* Cycle time of task calling TX and RX *)
	InitCAN3 := FALSE;											(* Execute this block one time for initialisation *)
END_IF	
IF (InitCAN4 = TRUE) THEN 
	CanInit(	iEnable			:= TRUE,                  		(* Initialiaze CAN *)
				iChannel		:= 4,							(* CAN Channel 4 *)
				iCAN			:= ADR(GVL.gCan4), 				(* Structure for sending / receiving CAN messages *)
				iBaudrate       := 250, 					    (* 250 kBit *)
				iCanIdExtended  := FALSE, 						(* Standard CAN Frame *)
				iEcuCycleTime  	:= T#10MS);						(* Cycle time of task calling TX and RX *)
	InitCAN4 := FALSE;											(* Execute this block one time for initialisation *)
END_IF	
IF (InitCAN5 = TRUE) THEN 
	CanInit(	iEnable			:= TRUE,                  		(* Initialiaze CAN *)
				iChannel		:= 5,							(* CAN Channel 5 *)
				iCAN			:= ADR(GVL.gCan5), 				(* Structure for sending / receiving CAN messages *)
				iBaudrate       := 250, 					    (* 500 kBit *)
				iCanIdExtended  := FALSE, 						(* Standard CAN Frame *)
				iEcuCycleTime  	:= T#10MS);						(* Cycle time of task calling TX and RX *)
	InitCAN5:= FALSE;											(* Execute this block one time for initialisation *)
END_IF				


(*UDC Sleep command*)
IF GVL.G_CMSleep = TRUE THEN
	GVL.G_tonCMSleep_timer(IN:=TRUE, PT:=T#5S);
	IF GVL.G_tonCMSleep_timer.Q THEN
		TTC_Sleep := TRUE;
	ELSE
		TTC_Sleep := FALSE;
	END_IF
ELSE
	GVL.G_tonCMSleep_timer(IN:=FALSE, PT:=T#5S);
	TTC_Sleep := FALSE;
END_IF

(*CAN Reveice*)
Receive_Msg();	

ChiefMaster(
	ssMethodType:= 1,
(*Inputs*)
(*Hardwired Inputs*)  
	AI_KL15:=DWORD_TO_REAL(WakeUp_mV),
	AI_HVIL_BDU:= DWORD_TO_REAL(AI_HVIL_BDU_P107), 
	AI_HVIL_Component:= DWORD_TO_REAL(AI_HVIL_Components_P108), 
	AI_HVIL_Battery:= DWORD_TO_REAL(AI_HVIL_Battery_P109),
	DI_HVIL_Overrule:= DI_HVIL_Overrule_P110, 
	AI_MainHV_Plus_FB:= DWORD_TO_REAL(AI_Main_Plus_FB_P115), 
	AI_MainHV_Minus_FB:= DWORD_TO_REAL(AI_Main_Minus_FB_P116), 
	AI_EmergencyButton_NC:= DWORD_TO_REAL(AI_EmergencyButton_NC_P131), 
	AI_EmergencyButton_NO:= DWORD_TO_REAL(KL15_mV), 
	DI_ResetButton_LED_NO:= DI_ResetButton_NO_P132, 
	DI_Proximity_BB1:= DI_Proximity_BB1_P133, 
	DI_Proximity_BB2:= DI_Proximity_BB2_P134, 
	DI_Proximity_BB3:= DI_Proximity_BB3_P135, 
	AI_DCHV_Plus_FB:= DWORD_TO_REAL(AI_DC_Plus_FB_P122), 
	AI_DCHV_Minus_FB:= DWORD_TO_REAL(AI_DC_Minus_FB_P123),
	DI_IMD_FB_BB1:= DI_IMD_FB_BB1_P112,
	DI_IMD_FB_BB2:= DI_IMD_FB_BB2_P113,
	DI_IMD_FB_BB3:= DI_IMD_FB_BB3_P114,
(*CAN Inputs*)	
	C_Actia_Batt1_MyStatus:= GVL.C_Actia_BB1_MyStatus, 
	C_Actia_Batt1_MyStatus_Timeout:= GVL.C_Actia_BB1_MyStatus_Timeout, 
	C_Actia_Batt1_Error:= GVL.C_Actia_BB1_Error, 
	C_Actia_Batt1_Error_Timeout:= GVL.C_Actia_BB1_Error_Timeout, 
	C_Actia_Batt1_ADS_8:= GVL.C_Actia_BB1_ADS_8, 
	C_Actia_Batt1_ADS_8_Timeout:= GVL.C_Actia_BB1_ADS_8_Timeout,
 	C_Actia_Batt1_ADS_0:= GVL.C_Actia_BB1_ADS_0, 
	C_Actia_Batt1_ADS_0_Timeout:= GVL.C_Actia_BB1_ADS_0_Timeout,
	C_Actia_Batt1_ADS_1:= GVL.C_Actia_BB1_ADS_1, 
	C_Actia_Batt1_ADS_1_Timeout:= GVL.C_Actia_BB1_ADS_1_Timeout, 
	C_Actia_Batt1_ADS_3:= GVL.C_Actia_BB1_ADS_3, 
	C_Actia_Batt1_ADS_3_Timeout:= GVL.C_Actia_BB1_ADS_3_Timeout, 
	C_Actia_Batt2_MyStatus:= GVL.C_Actia_BB2_MyStatus, 
	C_Actia_Batt2_MyStatus_Timeout:= GVL.C_Actia_BB2_MyStatus_Timeout, 
	C_Actia_Batt2_Error:= GVL.C_Actia_BB2_Error, 
	C_Actia_Batt2_Error_Timeout:= GVL.C_Actia_BB2_Error_Timeout, 
	C_Actia_Batt2_ADS_8:= GVL.C_Actia_BB2_ADS_8, 
	C_Actia_Batt2_ADS_8_Timeout:= GVL.C_Actia_BB2_ADS_8_Timeout,
  	C_Actia_Batt2_ADS_0:= GVL.C_Actia_BB2_ADS_0, 
	C_Actia_Batt2_ADS_0_Timeout:= GVL.C_Actia_BB2_ADS_0_Timeout,
	C_Actia_Batt2_ADS_1:= GVL.C_Actia_BB2_ADS_1, 
	C_Actia_Batt2_ADS_1_Timeout:= GVL.C_Actia_BB2_ADS_1_Timeout, 
	C_Actia_Batt2_ADS_3:= GVL.C_Actia_BB2_ADS_3, 
	C_Actia_Batt2_ADS_3_Timeout:= GVL.C_Actia_BB2_ADS_3_Timeout, 
	C_Actia_Batt3_MyStatus:= GVL.C_Actia_BB3_MyStatus, 
	C_Actia_Batt3_MyStatus_Timeout:= GVL.C_Actia_BB3_MyStatus_Timeout, 
	C_Actia_Batt3_Error:= GVL.C_Actia_BB3_Error,
	C_Actia_Batt3_Error_Timeout:= GVL.C_Actia_BB3_Error_Timeout, 
	C_Actia_Batt3_ADS_8:= GVL.C_Actia_BB3_ADS_8, 
	C_Actia_Batt3_ADS_8_Timeout:= GVL.C_Actia_BB3_ADS_8_Timeout,
  	C_Actia_Batt3_ADS_0:= GVL.C_Actia_BB3_ADS_0, 
	C_Actia_Batt3_ADS_0_Timeout:= GVL.C_Actia_BB3_ADS_0_Timeout,
	C_Actia_Batt3_ADS_1:= GVL.C_Actia_BB3_ADS_1, 
	C_Actia_Batt3_ADS_1_Timeout:= GVL.C_Actia_BB3_ADS_1_Timeout, 
	C_Actia_Batt3_ADS_3:= GVL.C_Actia_BB3_ADS_3, 
	C_Actia_Batt3_ADS_3_Timeout:= GVL.C_Actia_BB3_ADS_3_Timeout, 
	C_LB_Batt1_CellVoltage01_Msg:= GVL.C_LB_Batt1_CellVoltage01, 
	C_LB_Batt1_CellVoltage01_Timeout:= GVL.C_LB_Batt1_CellVoltage01_Timeout, 
	C_LB_Batt1_CellVoltage02_Msg:= GVL.C_LB_Batt1_CellVoltage02, 
	C_LB_Batt1_CellVoltage02_Timeout:= GVL.C_LB_Batt1_CellVoltage02_Timeout, 
	C_LB_Batt1_CellTemperature_Msg:= GVL.C_LB_Batt1_CellTemperature, 
	C_LB_Batt1_CellTemperature_Timeout:= GVL.C_LB_Batt1_CellTemperature_Timeout, 
	C_LB_Batt1_InsulationMonitor_Msg:= GVL.C_LB_Batt1_InsulationMonitor, 
	C_LB_Batt1_InsulationMonitor_Timeout:= GVL.C_LB_Batt1_InsulationMonitor_Timeout, 
	C_LB_Batt1_Status01_Msg:= GVL.C_LB_Batt1_Status01, 
	C_LB_Batt1_Status01_Timeout:= GVL.C_LB_Batt1_Status01_Timeout, 
	C_LB_BMS_Status02_Msg:= GVL.C_LB_Batt1_Status02, 
	C_LB_Batt1_Status02_Timeout:= GVL.C_LB_Batt1_Status02_Timeout, 
	C_LB_Batt1_Status03_Msg:= GVL.C_LB_Batt1_Status03, 
	C_LB_Batt1_Status03_Timeout:= GVL.C_LB_Batt1_Status03_Timeout, 
	C_LB_Batt2_CellVoltage01_Msg:= GVL.C_LB_Batt2_CellVoltage01, 
	C_LB_Batt2_CellVoltage01_Timeout:= GVL.C_LB_Batt2_CellVoltage01_Timeout, 
	C_LB_Batt2_CellVoltage02_Msg:= GVL.C_LB_Batt2_CellVoltage02, 
	C_LB_Batt2_CellVoltage02_Timeout:= GVL.C_LB_Batt2_CellVoltage02_Timeout, 
	C_LB_Batt2_CellTemperature_Msg:= GVL.C_LB_Batt2_CellTemperature, 
	C_LB_Batt2_CellTemperature_Timeout:= GVL.C_LB_Batt2_CellTemperature_Timeout, 
	C_LB_Batt2_InsulationMonitor_Msg:= GVL.C_LB_Batt2_InsulationMonitor, 
	C_LB_Batt2_InsulationMonitor_Timeout:= GVL.C_LB_Batt2_InsulationMonitor_Timeout, 
	C_LB_Batt2_Status01_Msg:= GVL.C_LB_Batt2_Status01, 
	C_LB_Batt2_Status01_Timeout:= GVL.C_LB_Batt2_Status01_Timeout, 
	C_LB_Batt2_Status02_Msg:= GVL.C_LB_Batt2_Status02, 
	C_LB_Batt2_Status02_Timeout:= GVL.C_LB_Batt2_Status02_Timeout, 
	C_LB_Batt2_Status03_Msg:= GVL.C_LB_Batt2_Status03, 
	C_LB_Batt2_Status03_Timeout:= GVL.C_LB_Batt2_Status03_Timeout, 
	C_LB_Batt3_CellVoltage01_Msg:= GVL.C_LB_Batt3_CellVoltage01, 
	C_LB_Batt3_CellVoltage01_Timeout:= GVL.C_LB_Batt3_CellVoltage01_Timeout, 
	C_LB_Batt3_CellVoltage02_Msg:= GVL.C_LB_Batt3_CellVoltage02, 
	C_LB_Batt3_CellVoltage02_Timeout:= GVL.C_LB_Batt3_CellVoltage02_Timeout, 
	C_LB_Batt3_CellTemperature_Msg:= GVL.C_LB_Batt3_CellTemperature, 
	C_LB_Batt3_CellTemperature_Timeout:= GVL.C_LB_Batt3_CellTemperature_Timeout, 
	C_LB_Batt3_InsulationMonitor_Msg:= GVL.C_LB_Batt3_InsulationMonitor, 
	C_LB_Batt3_InsulationMonitor_Timeout:= GVL.C_LB_Batt3_InsulationMonitor_Timeout, 
	C_LB_Batt3_Status01_Msg:= GVL.C_LB_Batt3_Status01, 
	C_LB_Batt3_Status01_Timeout:= GVL.C_LB_Batt3_Status01_Timeout, 
	C_LB_Batt3_Status02_Msg:= GVL.C_LB_Batt3_Status02, 
	C_LB_Batt3_Status02_Timeout:= GVL.C_LB_Batt3_Status02_Timeout, 
	C_LB_Batt3_Status03_Msg:= GVL.C_LB_Batt3_Status03, 
	C_LB_Batt3_Status03_Timeout:= GVL.C_LB_Batt3_Status03_Timeout, 
	C_UDC_Msg1:= GVL.C_UDC_Msg1, 
	C_UDC_Msg1_Timeout:= GVL.C_UDC_Msg1_Timeout,

	
(*Outputs*) 
(*HW Outputs*)
	CMSleep=> GVL.G_CMSleep, 
	DO_KL15_BB1=> DO_KL15_BB1_P149, 
	DO_KL15_BB2=> DO_KL15_BB2_P152, 
	DO_KL15_BB3=> DO_KL15_BB3_P155, 
	DO_REQ_MainHV_ON_MINUS=> DO_Request_Main_Minus_P239, 
	DO_REQ_MainHV_ON_PLUS=> DO_Request_Main_Plus_P238, 
	DO_REQ_MainHV_ON_Precharge=> DO_Request_Main_Precharge_P251,
 	DO_REQ_DC_ON_MINUS=> DO_Request_DC_Minus_P241,
	DO_REQ_DC_ON_PLUS=> DO_Request_DC_Plus_P240,
	DO_boKL15_IMD_BB1=> DO_IMD_BB1_P173,
	DO_boKL15_IMD_BB2=> DO_IMD_BB2_P176,
	DO_boKL15_IMD_BB3=> DO_IMD_BB3_P179,
	DO_CabinAlarm=> DO_CabinAlarm_P188,
	DO_boEMSRET_BDU1=> DO_EMSRET_BDU1, 
	DO_boEMSRET_BDU2=> DO_EMSRET_BDU2, 
	DO_boEMSRET_BB1_1=> DO_EMSRET_BB1_1, 
	DO_boEMSRET_BB1_2=> DO_EMSRET_BB1_2, 
	DO_boEMSRET_BB2_1=> DO_EMSRET_BB2_1, 
	DO_boEMSRET_BB2_2=> DO_EMSRET_BB2_2, 
	DO_boEMSRET_BB3_1=> DO_EMSRET_BB3_1, 
	DO_boEMSRET_BB3_2=> DO_EMSRET_BB3_2, 
	DO_HVIL_Supply=> DO_HVIL_Supply_P161,
	do_boResetButton_LED=> DO_REsetButton_LED_P185,
(*CAN Outputs*)	
	BMS_Control_Batt1=> GVL.C_Actia_Control_Batt1, 
	BMS_Control_Batt2=> GVL.C_Actia_Control_Batt2, 
	BMS_Control_Batt3=> GVL.C_Actia_Control_Batt3, 
	OP_LiBa_OperationRequest_Batt1=> GVL.C_LiBa_OperationRequest_Batt1, 
	OP_LiBa_OperationRequest_Batt2=> GVL.C_LiBa_OperationRequest_Batt2, 
	OP_LiBa_OperationRequest_Batt3=> GVL.C_LiBa_OperationRequest_Batt3, 
	OP_ChiefMaster_IP_Msg1=> GVL.C_Chief_Master_Msg1, 
	OP_ChiefMaster_OP_Msg2=> GVL.C_Chief_Master_Msg2, 
	OP_ChiefMaster_SS1_Msg3=> GVL.C_Chief_Master_Msg3, 
	OP_ChiefMaster_SS2_Msg4=> GVL.C_Chief_Master_Msg4, 
	OP_ChiefMaster_Calc_Msg5=> GVL.C_Chief_Master_Msg5, 
	OP_ChiefMaster_BDU_Msg6=> GVL.C_Chief_Master_Msg6, 
	OP_ChiefMaster_Battery1_Msg7=> GVL.C_Chief_Master_Msg7, 
	OP_ChiefMaster_Battery1_Msg8=> GVL.C_Chief_Master_Msg8, 
	OP_ChiefMaster_Battery1_Msg9=> GVL.C_Chief_Master_Msg9, 
	OP_ChiefMaster_Battery2_Msg10=> GVL.C_Chief_Master_Msg10, 
	OP_ChiefMaster_Battery2_Msg11=> GVL.C_Chief_Master_Msg11, 
	OP_ChiefMaster_Battery2_Msg12=> GVL.C_Chief_Master_Msg12,
	OP_ChiefMaster_Battery3_Msg13=> GVL.C_Chief_Master_Msg13,
	OP_ChiefMaster_Battery3_Msg14=> GVL.C_Chief_Master_Msg14,
	OP_ChiefMaster_Battery3_Msg15=> GVL.C_Chief_Master_Msg15);
	

(*CAN Send*)	
Transmit_Msg();

END_PROGRAM

// Device/Application/ChiefMaster
FUNCTION_BLOCK ChiefMaster
VAR_INPUT
	ssMethodType: SINT;
	AI_KL15: REAL;
	AI_HVIL_BDU: REAL;
	AI_HVIL_Component: REAL;
	AI_HVIL_Battery: REAL;
	DI_HVIL_Overrule: BOOL;
	AI_MainHV_Plus_FB: REAL;
	AI_MainHV_Minus_FB: REAL;
	AI_EmergencyButton_NC: REAL;
	AI_EmergencyButton_NO: REAL;
	DI_ResetButton_LED_NO: BOOL;
	DI_Proximity_BB1: BOOL;
	DI_Proximity_BB2: BOOL;
	DI_Proximity_BB3: BOOL;
	AI_DCHV_Plus_FB: REAL;
	AI_DCHV_Minus_FB: REAL;
	DI_IMD_FB_BB1: BOOL;
	DI_IMD_FB_BB2: BOOL;
	DI_IMD_FB_BB3: BOOL;
	C_Actia_Batt1_MyStatus: ARRAY[0..7] OF BYTE;
	C_Actia_Batt1_MyStatus_Timeout: BOOL;
	C_Actia_Batt1_Error: ARRAY[0..7] OF BYTE;
	C_Actia_Batt1_Error_Timeout: BOOL;
	C_Actia_Batt1_ADS_8: ARRAY[0..7] OF BYTE;
	C_Actia_Batt1_ADS_8_Timeout: BOOL;
	C_Actia_Batt1_ADS_0: ARRAY[0..7] OF BYTE;
	C_Actia_Batt1_ADS_0_Timeout: BOOL;
	C_Actia_Batt1_ADS_1: ARRAY[0..7] OF BYTE;
	C_Actia_Batt1_ADS_1_Timeout: BOOL;
	C_Actia_Batt1_ADS_3: ARRAY[0..7] OF BYTE;
	C_Actia_Batt1_ADS_3_Timeout: BOOL;
	C_Actia_Batt2_MyStatus: ARRAY[0..7] OF BYTE;
	C_Actia_Batt2_MyStatus_Timeout: BOOL;
	C_Actia_Batt2_Error: ARRAY[0..7] OF BYTE;
	C_Actia_Batt2_Error_Timeout: BOOL;
	C_Actia_Batt2_ADS_8: ARRAY[0..7] OF BYTE;
	C_Actia_Batt2_ADS_8_Timeout: BOOL;
	C_Actia_Batt2_ADS_0: ARRAY[0..7] OF BYTE;
	C_Actia_Batt2_ADS_0_Timeout: BOOL;
	C_Actia_Batt2_ADS_1: ARRAY[0..7] OF BYTE;
	C_Actia_Batt2_ADS_1_Timeout: BOOL;
	C_Actia_Batt2_ADS_3: ARRAY[0..7] OF BYTE;
	C_Actia_Batt2_ADS_3_Timeout: BOOL;
	C_Actia_Batt3_MyStatus: ARRAY[0..7] OF BYTE;
	C_Actia_Batt3_MyStatus_Timeout: BOOL;
	C_Actia_Batt3_Error: ARRAY[0..7] OF BYTE;
	C_Actia_Batt3_Error_Timeout: BOOL;
	C_Actia_Batt3_ADS_8: ARRAY[0..7] OF BYTE;
	C_Actia_Batt3_ADS_8_Timeout: BOOL;
	C_Actia_Batt3_ADS_0: ARRAY[0..7] OF BYTE;
	C_Actia_Batt3_ADS_0_Timeout: BOOL;
	C_Actia_Batt3_ADS_1: ARRAY[0..7] OF BYTE;
	C_Actia_Batt3_ADS_1_Timeout: BOOL;
	C_Actia_Batt3_ADS_3: ARRAY[0..7] OF BYTE;
	C_Actia_Batt3_ADS_3_Timeout: BOOL;
	C_LB_Batt1_CellVoltage01_Msg: ARRAY[0..7] OF BYTE;
	C_LB_Batt1_CellVoltage01_Timeout: BOOL;
	C_LB_Batt1_CellVoltage02_Msg: ARRAY[0..7] OF BYTE;
	C_LB_Batt1_CellVoltage02_Timeout: BOOL;
	C_LB_Batt1_CellTemperature_Msg: ARRAY[0..7] OF BYTE;
	C_LB_Batt1_CellTemperature_Timeout: BOOL;
	C_LB_Batt1_InsulationMonitor_Msg: ARRAY[0..7] OF BYTE;
	C_LB_Batt1_InsulationMonitor_Timeout: BOOL;
	C_LB_Batt1_Status01_Msg: ARRAY[0..7] OF BYTE;
	C_LB_Batt1_Status01_Timeout: BOOL;
	C_LB_BMS_Status02_Msg: ARRAY[0..7] OF BYTE;
	C_LB_Batt1_Status02_Timeout: BOOL;
	C_LB_Batt1_Status03_Msg: ARRAY[0..7] OF BYTE;
	C_LB_Batt1_Status03_Timeout: BOOL;
	C_LB_Batt2_CellVoltage01_Msg: ARRAY[0..7] OF BYTE;
	C_LB_Batt2_CellVoltage01_Timeout: BOOL;
	C_LB_Batt2_CellVoltage02_Msg: ARRAY[0..7] OF BYTE;
	C_LB_Batt2_CellVoltage02_Timeout: BOOL;
	C_LB_Batt2_CellTemperature_Msg: ARRAY[0..7] OF BYTE;
	C_LB_Batt2_CellTemperature_Timeout: BOOL;
	C_LB_Batt2_InsulationMonitor_Msg: ARRAY[0..7] OF BYTE;
	C_LB_Batt2_InsulationMonitor_Timeout: BOOL;
	C_LB_Batt2_Status01_Msg: ARRAY[0..7] OF BYTE;
	C_LB_Batt2_Status01_Timeout: BOOL;
	C_LB_Batt2_Status02_Msg: ARRAY[0..7] OF BYTE;
	C_LB_Batt2_Status02_Timeout: BOOL;
	C_LB_Batt2_Status03_Msg: ARRAY[0..7] OF BYTE;
	C_LB_Batt2_Status03_Timeout: BOOL;
	C_LB_Batt3_CellVoltage01_Msg: ARRAY[0..7] OF BYTE;
	C_LB_Batt3_CellVoltage01_Timeout: BOOL;
	C_LB_Batt3_CellVoltage02_Msg: ARRAY[0..7] OF BYTE;
	C_LB_Batt3_CellVoltage02_Timeout: BOOL;
	C_LB_Batt3_CellTemperature_Msg: ARRAY[0..7] OF BYTE;
	C_LB_Batt3_CellTemperature_Timeout: BOOL;
	C_LB_Batt3_InsulationMonitor_Msg: ARRAY[0..7] OF BYTE;
	C_LB_Batt3_InsulationMonitor_Timeout: BOOL;
	C_LB_Batt3_Status01_Msg: ARRAY[0..7] OF BYTE;
	C_LB_Batt3_Status01_Timeout: BOOL;
	C_LB_Batt3_Status02_Msg: ARRAY[0..7] OF BYTE;
	C_LB_Batt3_Status02_Timeout: BOOL;
	C_LB_Batt3_Status03_Msg: ARRAY[0..7] OF BYTE;
	C_LB_Batt3_Status03_Timeout: BOOL;
	C_UDC_Msg1: ARRAY[0..7] OF BYTE;
	C_UDC_Msg1_Timeout: BOOL;
END_VAR
VAR_OUTPUT
	CMSleep: BOOL;
	DO_KL15_BB1: BOOL;
	DO_KL15_BB2: BOOL;
	DO_KL15_BB3: BOOL;
	DO_REQ_MainHV_ON_MINUS: BOOL;
	DO_REQ_MainHV_ON_PLUS: BOOL;
	DO_REQ_MainHV_ON_Precharge: BOOL;
	DO_REQ_DC_ON_MINUS: BOOL;
	DO_REQ_DC_ON_PLUS: BOOL;
	DO_boKL15_IMD_BB1: BOOL;
	DO_boKL15_IMD_BB2: BOOL;
	DO_boKL15_IMD_BB3: BOOL;
	DO_CabinAlarm: BOOL;
	DO_boEMSRET_BDU1: BOOL;
	DO_boEMSRET_BDU2: BOOL;
	DO_boEMSRET_BB1_1: BOOL;
	DO_boEMSRET_BB1_2: BOOL;
	DO_boEMSRET_BB2_1: BOOL;
	DO_boEMSRET_BB2_2: BOOL;
	DO_boEMSRET_BB3_1: BOOL;
	DO_boEMSRET_BB3_2: BOOL;
	DO_HVIL_Supply: BOOL;
	DO_boResetButton_LED: BOOL;
	BMS_Control_Batt1: ARRAY[0..7] OF BYTE;
	BMS_Control_Batt2: ARRAY[0..7] OF BYTE;
	BMS_Control_Batt3: ARRAY[0..7] OF BYTE;
	OP_LiBa_OperationRequest_Batt1: ARRAY[0..7] OF BYTE;
	OP_LiBa_OperationRequest_Batt2: ARRAY[0..7] OF BYTE;
	OP_LiBa_OperationRequest_Batt3: ARRAY[0..7] OF BYTE;
	OP_ChiefMaster_IP_Msg1: ARRAY[0..7] OF BYTE;
	OP_ChiefMaster_OP_Msg2: ARRAY[0..7] OF BYTE;
	OP_ChiefMaster_SS1_Msg3: ARRAY[0..7] OF BYTE;
	OP_ChiefMaster_SS2_Msg4: ARRAY[0..7] OF BYTE;
	OP_ChiefMaster_Calc_Msg5: ARRAY[0..7] OF BYTE;
	OP_ChiefMaster_BDU_Msg6: ARRAY[0..7] OF BYTE;
	OP_ChiefMaster_Battery1_Msg7: ARRAY[0..7] OF BYTE;
	OP_ChiefMaster_Battery1_Msg8: ARRAY[0..7] OF BYTE;
	OP_ChiefMaster_Battery1_Msg9: ARRAY[0..7] OF BYTE;
	OP_ChiefMaster_Battery2_Msg10: ARRAY[0..7] OF BYTE;
	OP_ChiefMaster_Battery2_Msg11: ARRAY[0..7] OF BYTE;
	OP_ChiefMaster_Battery2_Msg12: ARRAY[0..7] OF BYTE;
	OP_ChiefMaster_Battery3_Msg13: ARRAY[0..7] OF BYTE;
	OP_ChiefMaster_Battery3_Msg14: ARRAY[0..7] OF BYTE;
	OP_ChiefMaster_Battery3_Msg15: ARRAY[0..7] OF BYTE;
END_VAR
VAR
	IP_boEV_IsolationMeasurementRequest: BOOL;
	IP_boChargeStop_Button: BOOL;
	boOutput_c: BOOL;
	IP_boKL15_D: BOOL;
	IP_boKL15_C: BOOL;
	IP_boBatt1_SDERR_activ: BOOL;
	IP_boBatt2_SDERR_activ: BOOL;
	IP_boBatt3_SDERR_activ: BOOL;
	IP_boBatt1_HV_REL_ON: BOOL;
	IP_boBatt2_HV_REL_ON: BOOL;
	IP_boBatt3_HV_REL_ON: BOOL;
	IP_boBatt1_HV_relay_MINUS_Sense: BOOL;
	IP_boBatt1_HV_relay_PLUS_Sense: BOOL;
	IP_boBatt2_HV_relay_MINUS_Sense: BOOL;
	IP_boBatt2_HV_relay_PLUS_Sense: BOOL;
	IP_boBatt3_HV_relay_MINUS_Sense: BOOL;
	IP_boBatt3_HV_relay_PLUS_Sense: BOOL;
	IP_boBatt1_Insulation_ready_and_OK: BOOL;
	IP_boBatt2_Insulation_ready_and_OK: BOOL;
	IP_boBatt3_Insulation_ready_and_OK: BOOL;
	IP_boBatt1_IMD_active: BOOL;
	IP_boBatt2_IMD_active: BOOL;
	IP_boBatt3_IMD_active: BOOL;
	REQ_HV_ON_a: LREAL;
	REQ_HV_ON_d: LREAL;
	REQ_HV_ON: LREAL;
	IP_boSafeToShutdown: BOOL;
	boOutput_n: BOOL;
	boOutput_h: BOOL;
	boOutput_k: BOOL;
	b_Constant: UINT;
	Constant_n: UINT;
	Constant_o: UINT;
	boOutput_o: BOOL;
	boOutput_a: BOOL;
	boOutput: BOOL;
	clockTickCounter: DINT;
	ShiftArithmetic6: USINT;
	ShiftArithmetic5: USINT;
	ShiftArithmetic4: USINT;
	ShiftArithmetic2: USINT;
	ShiftArithmetic: USINT;
	ShiftArithmetic6_a: USINT;
	ShiftArithmetic5_j: USINT;
	ShiftArithmetic4_h: USINT;
	ShiftArithmetic3: USINT;
	ShiftArithmetic2_c: USINT;
	ShiftArithmetic_n: USINT;
	ShiftArithmetic6_f: USINT;
	ShiftArithmetic5_h: USINT;
	ShiftArithmetic2_o: USINT;
	ShiftArithmetic5_jh: USINT;
	ShiftArithmetic2_n: USINT;
	ShiftArithmetic5_f: USINT;
	ShiftArithmetic2_h: USINT;
	ShiftArithmetic4_m: USINT;
	ShiftArithmetic2_k: USINT;
	ShiftArithmetic_m: USINT;
	ShiftArithmetic6_i: USINT;
	ShiftArithmetic5_k: USINT;
	ShiftArithmetic6_m: USINT;
	ShiftArithmetic5_a: USINT;
	ShiftArithmetic4_a: USINT;
	ShiftArithmetic3_k: USINT;
	ShiftArithmetic2_p: USINT;
	ShiftArithmetic6_h: USINT;
	ShiftArithmetic4_n: USINT;
	ShiftArithmetic2_d: USINT;
	ShiftArithmetic6_n: USINT;
	ShiftArithmetic5_a2: USINT;
	ShiftArithmetic3_o: USINT;
	ShiftArithmetic2_b: USINT;
	ShiftArithmetic6_k: USINT;
	ShiftArithmetic5_i: USINT;
	ShiftArithmetic4_ap: USINT;
	ShiftArithmetic3_e: USINT;
	ShiftArithmetic1: USINT;
	ShiftArithmetic_h: USINT;
	ShiftArithmetic6_kx: USINT;
	ShiftArithmetic5_ke: USINT;
	ShiftArithmetic4_d: USINT;
	ShiftArithmetic3_oe: USINT;
	ShiftArithmetic2_ot: USINT;
	ShiftArithmetic1_n: USINT;
	ShiftArithmetic6_kxt: USINT;
	ShiftArithmetic5_hi: USINT;
	ShiftArithmetic4_b: USINT;
	ShiftArithmetic3_o0: USINT;
	ShiftArithmetic2_e: USINT;
	ShiftArithmetic1_nm: USINT;
	ShiftArithmetic6_b: USINT;
	ShiftArithmetic5_b: USINT;
	ShiftArithmetic4_p: USINT;
	ShiftArithmetic3_a: USINT;
	ShiftArithmetic2_m: USINT;
	ShiftArithmetic1_nx: USINT;
	ShiftArithmetic6_ap: USINT;
	ShiftArithmetic5_m: USINT;
	ShiftArithmetic4_l: USINT;
	ShiftArithmetic3_h: USINT;
	ShiftArithmetic2_f: USINT;
	ShiftArithmetic_k: USINT;
	DataTypeConversion3: USINT;
	ShiftArithmetic6_o: USINT;
	ShiftArithmetic5_k0: USINT;
	ShiftArithmetic4_f: USINT;
	ShiftArithmetic3_l: USINT;
	ShiftArithmetic2_fl: USINT;
	ShiftArithmetic_a: USINT;
	DataTypeConversion3_d: USINT;
	ShiftArithmetic6_mw: USINT;
	ShiftArithmetic5_c: USINT;
	ShiftArithmetic4_db: USINT;
	ShiftArithmetic3_c: USINT;
	ShiftArithmetic2_g: USINT;
	ShiftArithmetic_p: USINT;
	DataTypeConversion3_l: USINT;
	Subsystem1_MODE: BOOL;
	Subsystem_MODE_dz: BOOL;
	Subsystem_MODE_d: BOOL;
	Subsystem_MODE_e: BOOL;
	Subsystem_MODE_h: BOOL;
	Subsystem_MODE_c: BOOL;
	Subsystem_MODE: BOOL;
	IP_boEVDisconnectingDevice: BOOL;
	IP_boBatt1_ERROR_activ: BOOL;
	IP_boBatt1_WARNING_activ: BOOL;
	IP_boBatt2_ERROR_activ: BOOL;
	IP_boBatt2_WARNING_activ: BOOL;
	IP_boBatt3_ERROR_activ: BOOL;
	IP_boBatt3_WARNING_activ: BOOL;
	UnitDelay1_DSTATE_f: LREAL;
	UnitDelay_DSTATE_o: LREAL;
	UnitDelay3_DSTATE_p: LREAL;
	UnitDelay2_DSTATE_a: LREAL;
	UnitDelay1_DSTATE_b: BOOL;
	UnitDelay_DSTATE_h: REAL;
	UnitDelay_DSTATE_i: USINT;
	REQ_MainHV_ON_MINUS: BOOL;
	REQ_MainHV_ON_MINUS_g: BOOL;
	REQ_MainHV_ON_PLUS: BOOL;
	is_active_c19_ChiefMaster: USINT;
	is_c19_ChiefMaster: USINT;
	is_c4_ChiefMaster: USINT;
	temporalCounter_i1_m: PLC_CODER_TIMER;
	is_active_c4_ChiefMaster: USINT;
	is_active_c46_ChiefMaster: USINT;
	is_c46_ChiefMaster: USINT;
	MainHV_Minus_Status: LREAL;
	is_c40_ChiefMaster: USINT;
	temporalCounter_i1_k: PLC_CODER_TIMER;
	is_active_c40_ChiefMaster: USINT;
	MainHV_Plus_Status: LREAL;
	is_c41_ChiefMaster: USINT;
	temporalCounter_i1_he: PLC_CODER_TIMER;
	is_active_c41_ChiefMaster: USINT;
	is_c53_ChiefMaster: USINT;
	temporalCounter_i1_n: PLC_CODER_TIMER;
	is_active_c53_ChiefMaster: USINT;
	is_c54_ChiefMaster: USINT;
	temporalCounter_i1_a: PLC_CODER_TIMER;
	is_active_c54_ChiefMaster: USINT;
	is_c51_ChiefMaster: USINT;
	temporalCounter_i1_h: PLC_CODER_TIMER;
	is_active_c51_ChiefMaster: USINT;
	is_active_c49_ChiefMaster: USINT;
	is_c49_ChiefMaster: USINT;
	temporalCounter_i1: PLC_CODER_TIMER;
	UnitDelay_DSTATE: LREAL;
	UnitDelay6_DSTATE: LREAL;
	UnitDelay1_DSTATE: LREAL;
	UnitDelay7_DSTATE: LREAL;
	UnitDelay2_DSTATE: LREAL;
	UnitDelay8_DSTATE: LREAL;
	UnitDelay5_DSTATE: LREAL;
	UnitDelay4_DSTATE: LREAL;
	UnitDelay3_DSTATE: LREAL;
	REQ_HV_Open_Batt1: BOOL;
	UnitDelay2_DSTATE_d: BOOL;
	REQ_HV_Open_Batt2: BOOL;
	UnitDelay6_DSTATE_b: BOOL;
	REQ_HV_Open_Batt3: BOOL;
	UnitDelay7_DSTATE_j: BOOL;
	System_Error: BOOL;
	UnitDelay9_DSTATE: BOOL;
	UnitDelay1_DSTATE_fl: BOOL;
	UnitDelay2_DSTATE_g: BOOL;
	UnitDelay6_DSTATE_h: BOOL;
	UnitDelay5_DSTATE_e: LREAL;
	FL_sST_MaxChargeCurrent: REAL;
	UnitDelay_DSTATE_d: BOOL;
	UnitDelay1_DSTATE_m: BOOL;
	UnitDelay2_DSTATE_m: BOOL;
	DelayInput1_DSTATE: LREAL;
	WeldingDetection_Status: USINT;
	DelayInput1_DSTATE_g: BOOL;
	DelayInput1_DSTATE_n: BOOL;
	DelayInput1_DSTATE_e: BOOL;
	UnitDelay4_DSTATE_n: BOOL;
	UnitDelay1_DSTATE_l: LREAL;
	UnitDelay9_DSTATE_d: BOOL;
	UnitDelay8_DSTATE_k: BOOL;
	UnitDelay7_DSTATE_h: BOOL;
	DataTypeConversion1: USINT;
	DataTypeConversion2: USINT;
	DataTypeConversion4: USINT;
	DataTypeConversion5: USINT;
	DataTypeConversion6: USINT;
	DataTypeConversion7: USINT;
	DataTypeConversion1_l: USINT;
	DataTypeConversion2_b: USINT;
	DataTypeConversion4_l: USINT;
	DataTypeConversion5_k: USINT;
	DataTypeConversion6_e: USINT;
	DataTypeConversion7_p: USINT;
	DataTypeConversion1_o: USINT;
	DataTypeConversion2_o: USINT;
	DataTypeConversion4_i: USINT;
	DataTypeConversion5_n: USINT;
	DataTypeConversion6_k: USINT;
	DataTypeConversion7_pe: USINT;
	DataTypeConversion6_h: USINT;
	DataTypeConversion6_p: USINT;
	DataTypeConversion6_l: USINT;
	ExtractDesiredBits: USINT;
	ExtractDesiredBits_m: USINT;
	ExtractDesiredBits_n: USINT;
	ExtractDesiredBits_b: USINT;
	ExtractDesiredBits_m1: USINT;
	ExtractDesiredBits_p: USINT;
	DataTypeConversion_c: USINT;
	DataTypeConversion_i: USINT;
	DataTypeConversion: USINT;
	ContactorState_i: LREAL;
	ContactorState_f: LREAL;
	ContactorState: LREAL;
	Precharge_Satus: LREAL;
	BatteryReadyToShutDown: BOOL;
	MainHV_Minus_Welded: BOOL;
	MainHV_Plus_Welded: BOOL;
	CMState_e2: USINT;
	boOutput_l: BOOL;
	boOutput_p: BOOL;
	boOutput_f: BOOL;
	Delay_DSTATE: ARRAY[0..2] OF BOOL;
	Delay_DSTATE_o: ARRAY[0..2] OF BOOL;
	Delay_DSTATE_k: ARRAY[0..2] OF BOOL;
	Delay_DSTATE_a: ARRAY[0..2] OF BOOL;
	Delay_DSTATE_ov: ARRAY[0..2] OF BOOL;
	Delay_DSTATE_c: ARRAY[0..2] OF BOOL;
	i0_Chart_m: Chart_m;
	i1_Chart_m: Chart_m;
	i2_Chart_m: Chart_m;
	i0_ChartBatt1: ChartBatt1;
	i0_Chartbatt2: Chartbatt2;
	i0_ChartBatt3: ChartBatt3;
	i0_Lib_InputProcessing_state: Lib_InputProcessing_state;
	i1_Lib_InputProcessing_state: Lib_InputProcessing_state;
	i2_Lib_InputProcessing_state: Lib_InputProcessing_state;
	i2_IMD_OK: IMD_OK;
	i0_IMD_OK: IMD_OK;
	i1_IMD_OK: IMD_OK;
	i0_REQ_HV_ON_Batt: REQ_HV_ON_Batt;
	i0_Chart_PrechargeStatus: Chart_PrechargeStatus;
	i3_Chart_SetDominantSwitch: Chart_SetDominantSwitch;
	i0_EmergencySD: EmergencySD;
	i0_Input_Delay: Input_Delay;
	i1_Input_Delay: Input_Delay;
	i2_Input_Delay: Input_Delay;
	i0_SDError: SDError;
	i0_BattChargeFcn: BattChargeFcn;
	i0_Chart_REQ_MAIN_MINUS: Chart_REQ_MAIN_MINUS;
	i0_Chart_WeldingDetection: Chart_WeldingDetection;
	i0_InsulationMonitoringReq: InsulationMonitoringReq;
	i0_Chart_jj: Chart_jj;
	i0_Chart1: Chart1;
	i1_Chart_jj: Chart_jj;
	i1_Chart1: Chart1;
	i0_Chart_lg: Chart_lg;
	i0_Chart1_l: Chart1_l;
	i1_Chart_lg: Chart_lg;
	i1_Chart1_l: Chart1_l;
	i2_Chart_lg: Chart_lg;
	i2_Chart1_l: Chart1_l;
	i2_Chart_jj: Chart_jj;
	i2_Chart1: Chart1;
	i0_CMState: CMState;
	i0_EMSRET_Power: EMSRET_Power;
	i5_Chart_Hysteresis_HighActive: Chart_Hysteresis_HighActive;
	i0_IMDOK_Input_Delay: IMDOK_Input_Delay;
	i1_IMDOK_Input_Delay: IMDOK_Input_Delay;
	i2_IMDOK_Input_Delay: IMDOK_Input_Delay;
	i0_Chart_Hysteresis_LowActive: Chart_Hysteresis_LowActive;
	i0_Chart_Hysteresis_HighActive: Chart_Hysteresis_HighActive;
	i1_Chart_Hysteresis_HighActive: Chart_Hysteresis_HighActive;
	i2_Chart_Hysteresis_HighActive: Chart_Hysteresis_HighActive;
	i0_HVIL_Input_Delay: HVIL_Input_Delay;
	i3_Chart_Hysteresis_HighActive: Chart_Hysteresis_HighActive;
	i1_HVIL_Input_Delay: HVIL_Input_Delay;
	i4_Chart_Hysteresis_HighActive: Chart_Hysteresis_HighActive;
	i2_HVIL_Input_Delay: HVIL_Input_Delay;
	i2_Chart_Hysteresis_LowActive: Chart_Hysteresis_LowActive;
	i1_Chart_Hysteresis_LowActive: Chart_Hysteresis_LowActive;
	i3_Chart_Hysteresis_LowActive: Chart_Hysteresis_LowActive;
	i0_SafeToCloseHV: SafeToCloseHV;
	i0_VoltageDetermination: VoltageDetermination;
	maxV: REAL;
	rtb_IT_boUDC_EV_IsolationMeasurementRequest: BOOL;
	rtb_IT_boChargeStop_Button: BOOL;
	rtb_S_in: BOOL;
	rtb_FL_boCMSleep: BOOL;
	rtb_IT_boUDC_KL15_D: BOOL;
	rtb_IT_boUDC_KL15_C: BOOL;
	rtb_FL_boKL15_Disable: BOOL;
	rtb_IP_boBatt1_Actia_Availability: BOOL;
	rtb_BattSelect_f: LREAL;
	rtb_BattSelect: LREAL;
	rtb_BattSelect_i: LREAL;
	rtb_Switch2_d: BOOL;
	rtb_ExtractDesiredBits_b13: USINT;
	rtb_Delay_dl: BOOL;
	rtb_Delay_j: BOOL;
	rtb_out_l: BOOL;
	rtb_Add_psl: REAL;
	rtb_IT_boBMS_SDError_BB1: BOOL;
	rtb_UnitDelay5: DINT;
	rtb_FL_boSS_HVIL_NOK: BOOL;
	rtb_FL_boHVC_AllCellBalanced: BOOL;
	rtb_Contactor_FB_State_h: LREAL;
	rtb_Contactor_FB_State_g: LREAL;
	rtb_Contactor_FB_State: LREAL;
	rtb_Min: REAL;
	rtb_out_n: BOOL;
	rtb_Switch1_fj: BOOL;
	rtb_FL_boKL15_Reset: BOOL;
	rtb_boData_Out: BOOL;
	rtb_IT_sHW_EmergencyButton_NC: BOOL;
	rtb_IT_boHW_EmergencyButton_NO: BOOL;
	rtb_IT_boHW_HVIL_BDU: BOOL;
	rtb_Out: USINT;
	rtb_out_i: BOOL;
	rtb_out_ne: BOOL;
	rtb_AND_l2: BOOL;
	rtb_AND_ni: BOOL;
	rtb_AND_ma: BOOL;
	rtb_System_SD_ErrorCode: USINT;
	rtb_UnitDelay: REAL;
	rtb_Switch3: REAL;
	rtb_UnitDelay1_d: BOOL;
	rtb_FL_boSS_BDU_Reset: BOOL;
	rtb_Out_k: BOOL;
	rtb_Add_an: REAL;
	rtb_Add_ic: REAL;
	rtb_IT_boBMS_HV_ON_BB: BOOL;
	rtb_Switch_a: REAL;
	rtb_Switch2_k: REAL;
	rtb_Out_bl: BOOL;
	rtb_IMD_State_g: USINT;
	rtb_IMD_State: USINT;
	rtb_Out_ap: BOOL;
	rtb_Switch_b: BOOL;
	rtb_Uk1: LREAL;
	rtb_Add_e: REAL;
	rtb_Add_en: REAL;
	rtb_IP_boBMS_SDError_BB1: BOOL;
	rtb_IP_boBMS_SDError_BB2: BOOL;
	rtb_IP_boBMS_SDError_BB3: BOOL;
	rtb_Add_nm: REAL;
	rtb_IP_boBMS_HV_REL_ON_BB1: BOOL;
	rtb_Add_d4: REAL;
	rtb_IP_boBMS_HV_REL_ON_BB2: BOOL;
	rtb_Add_cw: REAL;
	rtb_IP_boBMS_HV_REL_ON_BB3: BOOL;
	rtb_Add_ki5: REAL;
	rtb_Add_ir: REAL;
	rtb_Add_m: REAL;
	rtb_Add_b: REAL;
	rtb_DataTypeConversion_k: USINT;
	rtb_DataTypeConversion1: USINT;
	rtb_DataTypeConversion2_h: USINT;
	rtb_Add_h: REAL;
	rtb_Add_g: REAL;
	rtb_Add_ic5: REAL;
	rtb_Add_kf: REAL;
	rtb_Add_j3: REAL;
	rtb_Add_cv: REAL;
	rtb_Add_d: REAL;
	rtb_Add_ky: REAL;
	rtb_Add_ci: REAL;
	rtb_Add_c0: REAL;
	rtb_Add_egs: REAL;
	rtb_IP_boBMS_HV_Minus_Sense_BB1: BOOL;
	rtb_IP_boBMS_HV_Plus_Sense_BB1: BOOL;
	rtb_IP_boBMS_HV_Minus_Sense_BB2: BOOL;
	rtb_IP_boBMS_HV_Plus_Sense_BB2: BOOL;
	rtb_IP_boBMS_HV_Minus_Sense_BB3: BOOL;
	rtb_IP_boBMS_HV_Plus_Sense_BB3: BOOL;
	rtb_Add_ie: REAL;
	rtb_Add_oy: REAL;
	rtb_Add_bh: REAL;
	rtb_Add_no: REAL;
	rtb_IP_boBMS_IMD_Active_BB1: BOOL;
	rtb_IP_boBMS_IMD_Active_BB2: BOOL;
	rtb_IP_boBMS_IMD_Active_BB3: BOOL;
	rtb_IP_boBMS_Batt1_Availability: DINT;
	rtb_IP_boBMS_Batt3_Availability: DINT;
	rtb_Add_a5: REAL;
	rtb_Add_g4: REAL;
	rtb_Add_i5o: REAL;
	rtb_Add_pi: REAL;
	rtb_Add_eo: REAL;
	rtb_IT_boBMS_Error_BB1: BOOL;
	rtb_IT_boBMS_Error_BB2: BOOL;
	rtb_IT_boBMS_Error_BB3: BOOL;
	rtb_IT_boBMS_Warning_BB1: BOOL;
	rtb_IT_boBMS_Warning_BB2: BOOL;
	rtb_IT_boBMS_Warning_BB3: BOOL;
	rtb_IT_sBMS_InternalResistance_BB1_ohms: REAL;
	rtb_Abs: REAL;
	rtb_Abs1: REAL;
	rtb_Abs2: REAL;
	rtb_Divide_i: REAL;
	rtb_Divide1_p: REAL;
	rtb_Divide2: REAL;
	rtb_UnitDelay2: LREAL;
	rtb_IT_boUDC_SafeToShutdown: BOOL;
	rtb_Add_kr: DINT;
	rtb_Switch5_bs: REAL;
	rtb_FL_sSS_MaxDisChargeCurrent: REAL;
	rtb_Divide_h: REAL;
	rtb_ExtractDesiredBits_be: USINT;
	rtb_IT_boHW_MainHV_Minus_FB: BOOL;
	rtb_FL_boSS_System_Error: BOOL;
	rtb_NOT_m5: BOOL;
	rtb_IT_boHW_MainHV_Plus_FB: BOOL;
	rtb_IT_boHW_DCHV_Minus_FB: BOOL;
	rtb_IT_boHW_DCHV_Plus_FB: BOOL;
	rtb_ExtractDesiredBits_mi: USINT;
	rtb_ExtractDesiredBits_ebk: USINT;
	rtb_ShiftArithmetic3_p: USINT;
	Count_k: LREAL;
	v: LREAL;
	y: LREAL;
	y_0: LREAL;
	y_1: REAL;
	rtb_ExtractDesiredBits_bk_tmp: USINT;
	v_tmp: LREAL;
	OP_ChiefMaster_Battery1_Msg7_tmp: UDINT;
	OP_ChiefMaster_Battery2_Msg10_tmp: UDINT;
	OP_ChiefMaster_Battery3_Msg13_tmp: UDINT;
	temp1: BOOL;
	temp2: BOOL;
	temp3: REAL;
	b_temp2: REAL;
	b_temp3: REAL;
	temp4: REAL;
	temp5: USINT;
END_VAR



CASE ssMethodType OF
    SS_INITIALIZE: 
        (* SystemInitialize for Atomic SubSystem: '<Root>/ChiefMaster' *)
        (* Start for Constant: '<S392>/Constant' *)
        b_Constant := USINT_TO_UINT(IP_u8HW_IN_delay_ms);
        (* Start for Constant: '<S393>/Constant' incorporates:
         *  Constant: '<S392>/Constant' *)
        Constant_n := USINT_TO_UINT(IP_u8HW_IN_delay_ms);
        (* Start for Constant: '<S394>/Constant' incorporates:
         *  Constant: '<S392>/Constant' *)
        Constant_o := USINT_TO_UINT(IP_u8HW_IN_delay_ms);
        (* InitializeConditions for UnitDelay: '<S10>/Unit Delay' *)
        UnitDelay_DSTATE := 0.0;
        (* InitializeConditions for UnitDelay: '<S10>/Unit Delay6' *)
        UnitDelay6_DSTATE := 0.0;
        (* InitializeConditions for UnitDelay: '<S10>/Unit Delay1' *)
        UnitDelay1_DSTATE := 0.0;
        (* InitializeConditions for UnitDelay: '<S10>/Unit Delay7' *)
        UnitDelay7_DSTATE := 0.0;
        (* InitializeConditions for UnitDelay: '<S10>/Unit Delay2' *)
        UnitDelay2_DSTATE := 0.0;
        (* InitializeConditions for UnitDelay: '<S10>/Unit Delay8' *)
        UnitDelay8_DSTATE := 0.0;
        (* InitializeConditions for Delay: '<S768>/Delay' *)
        Delay_DSTATE[0] := FALSE;
        (* InitializeConditions for Delay: '<S766>/Delay' *)
        Delay_DSTATE_o[0] := FALSE;
        (* InitializeConditions for Delay: '<S767>/Delay' *)
        Delay_DSTATE_k[0] := FALSE;
        (* InitializeConditions for Delay: '<S723>/Delay' *)
        Delay_DSTATE_a[0] := FALSE;
        (* InitializeConditions for Delay: '<S721>/Delay' *)
        Delay_DSTATE_ov[0] := FALSE;
        (* InitializeConditions for Delay: '<S722>/Delay' *)
        Delay_DSTATE_c[0] := FALSE;
        (* InitializeConditions for Delay: '<S768>/Delay' *)
        Delay_DSTATE[1] := FALSE;
        (* InitializeConditions for Delay: '<S766>/Delay' *)
        Delay_DSTATE_o[1] := FALSE;
        (* InitializeConditions for Delay: '<S767>/Delay' *)
        Delay_DSTATE_k[1] := FALSE;
        (* InitializeConditions for Delay: '<S723>/Delay' *)
        Delay_DSTATE_a[1] := FALSE;
        (* InitializeConditions for Delay: '<S721>/Delay' *)
        Delay_DSTATE_ov[1] := FALSE;
        (* InitializeConditions for Delay: '<S722>/Delay' *)
        Delay_DSTATE_c[1] := FALSE;
        (* InitializeConditions for Delay: '<S768>/Delay' *)
        Delay_DSTATE[2] := FALSE;
        (* InitializeConditions for Delay: '<S766>/Delay' *)
        Delay_DSTATE_o[2] := FALSE;
        (* InitializeConditions for Delay: '<S767>/Delay' *)
        Delay_DSTATE_k[2] := FALSE;
        (* InitializeConditions for Delay: '<S723>/Delay' *)
        Delay_DSTATE_a[2] := FALSE;
        (* InitializeConditions for Delay: '<S721>/Delay' *)
        Delay_DSTATE_ov[2] := FALSE;
        (* InitializeConditions for Delay: '<S722>/Delay' *)
        Delay_DSTATE_c[2] := FALSE;
        (* InitializeConditions for UnitDelay: '<S8>/Unit Delay5' *)
        UnitDelay5_DSTATE := 0.0;
        (* InitializeConditions for UnitDelay: '<S8>/Unit Delay4' *)
        UnitDelay4_DSTATE := 0.0;
        (* InitializeConditions for UnitDelay: '<S8>/Unit Delay3' *)
        UnitDelay3_DSTATE := 0.0;
        (* InitializeConditions for UnitDelay: '<S8>/Unit Delay2' *)
        UnitDelay2_DSTATE_d := FALSE;
        (* InitializeConditions for UnitDelay: '<S8>/Unit Delay6' *)
        UnitDelay6_DSTATE_b := FALSE;
        (* InitializeConditions for UnitDelay: '<S8>/Unit Delay7' *)
        UnitDelay7_DSTATE_j := FALSE;
        (* InitializeConditions for UnitDelay: '<S8>/Unit Delay9' *)
        UnitDelay9_DSTATE := FALSE;
        (* InitializeConditions for UnitDelay: '<S8>/Unit Delay1' *)
        UnitDelay1_DSTATE_fl := FALSE;
        (* InitializeConditions for UnitDelay: '<S35>/Unit Delay1' *)
        UnitDelay1_DSTATE_f := 0.0;
        (* InitializeConditions for UnitDelay: '<S35>/Unit Delay' *)
        UnitDelay_DSTATE_o := 0.0;
        (* InitializeConditions for UnitDelay: '<S35>/Unit Delay2' *)
        UnitDelay2_DSTATE_g := FALSE;
        (* InitializeConditions for UnitDelay: '<S13>/Unit Delay3' *)
        UnitDelay3_DSTATE_p := 0.0;
        (* InitializeConditions for UnitDelay: '<S13>/Unit Delay2' *)
        UnitDelay2_DSTATE_a := 0.0;
        (* InitializeConditions for UnitDelay: '<S13>/Unit Delay6' *)
        UnitDelay6_DSTATE_h := FALSE;
        (* InitializeConditions for UnitDelay: '<S13>/Unit Delay5' *)
        UnitDelay5_DSTATE_e := 0.0;
        (* InitializeConditions for UnitDelay: '<S13>/Unit Delay1' *)
        UnitDelay1_DSTATE_b := FALSE;
        (* InitializeConditions for UnitDelay: '<S110>/Unit Delay' *)
        UnitDelay_DSTATE_h := 1.0;
        (* InitializeConditions for UnitDelay: '<S121>/Unit Delay' *)
        UnitDelay_DSTATE_d := FALSE;
        (* InitializeConditions for UnitDelay: '<S121>/Unit Delay1' *)
        UnitDelay1_DSTATE_m := FALSE;
        (* InitializeConditions for UnitDelay: '<S121>/Unit Delay2' *)
        UnitDelay2_DSTATE_m := FALSE;
        (* InitializeConditions for UnitDelay: '<S29>/Delay Input1'
         *
         * Block description for '<S29>/Delay Input1':
         *  
         *  Store in Global RAM *)
        DelayInput1_DSTATE := 0.0;
        (* InitializeConditions for UnitDelay: '<S21>/Unit Delay' *)
        UnitDelay_DSTATE_i := 0;
        (* InitializeConditions for UnitDelay: '<S94>/Delay Input1'
         *
         * Block description for '<S94>/Delay Input1':
         *  
         *  Store in Global RAM *)
        DelayInput1_DSTATE_g := FALSE;
        (* InitializeConditions for UnitDelay: '<S99>/Delay Input1'
         *
         * Block description for '<S99>/Delay Input1':
         *  
         *  Store in Global RAM *)
        DelayInput1_DSTATE_n := FALSE;
        (* InitializeConditions for UnitDelay: '<S104>/Delay Input1'
         *
         * Block description for '<S104>/Delay Input1':
         *  
         *  Store in Global RAM *)
        DelayInput1_DSTATE_e := FALSE;
        (* InitializeConditions for UnitDelay: '<S12>/Unit Delay4' *)
        UnitDelay4_DSTATE_n := FALSE;
        (* InitializeConditions for UnitDelay: '<S12>/Unit Delay1' *)
        UnitDelay1_DSTATE_l := 0.0;
        (* InitializeConditions for UnitDelay: '<S122>/Unit Delay9' *)
        UnitDelay9_DSTATE_d := FALSE;
        (* InitializeConditions for UnitDelay: '<S122>/Unit Delay8' *)
        UnitDelay8_DSTATE_k := FALSE;
        (* InitializeConditions for UnitDelay: '<S122>/Unit Delay7' *)
        UnitDelay7_DSTATE_h := FALSE;
        (* InitializeConditions for DiscretePulseGenerator: '<S114>/Discrete Pulse Generator20' *)
        clockTickCounter := 0;
        (* SystemInitialize for Enabled SubSystem: '<S195>/Subsystem1' *)
        (* SystemInitialize for DataTypeConversion: '<S664>/Data Type Conversion2' incorporates:
         *  Outport: '<S664>/TTC_Status_Databus' *)
        IP_boSafeToShutdown := FALSE;
        (* SystemInitialize for DataTypeConversion: '<S664>/Data Type Conversion3' incorporates:
         *  Outport: '<S664>/TTC_Status_Databus' *)
        IP_boKL15_D := FALSE;
        (* SystemInitialize for DataTypeConversion: '<S664>/Data Type Conversion4' incorporates:
         *  Outport: '<S664>/TTC_Status_Databus' *)
        IP_boKL15_C := FALSE;
        (* SystemInitialize for DataTypeConversion: '<S664>/Data Type Conversion5' incorporates:
         *  Outport: '<S664>/TTC_Status_Databus' *)
        IP_boEVDisconnectingDevice := FALSE;
        (* SystemInitialize for SignalConversion: '<S664>/TmpBufferAtConstantOutport1' incorporates:
         *  Outport: '<S664>/TTC_Status_Databus' *)
        IP_boEV_IsolationMeasurementRequest := FALSE;
        (* SystemInitialize for DataTypeConversion: '<S664>/Data Type Conversion7' incorporates:
         *  Outport: '<S664>/TTC_Status_Databus' *)
        IP_boChargeStop_Button := FALSE;
        (* End of SystemInitialize for SubSystem: '<S195>/Subsystem1' *)
        (* End of SystemInitialize for SubSystem: '<Root>/ChiefMaster' *)
        

        (* Constant: '<S387>/Constant4' incorporates:
         *  Constant: '<S387>/Constant'
         *  Constant: '<S387>/Constant1'
         *  Constant: '<S387>/Constant2'
         *  Constant: '<S387>/Constant3' *)
        i5_Chart_Hysteresis_HighActive(ssMethodType := SS_INITIALIZE, sSignal := AI_KL15, boInitial_Value := FALSE, boValue_Activated := TRUE, boValue_Deactivated := FALSE, sLB := 18000.0, b_sUB := 22000.0);
        boOutput_c := i5_Chart_Hysteresis_HighActive.boOutput;
        (* Outport: '<Root>/DO_KL15_BB1' *)
        i0_Chart_m(ssMethodType := SS_INITIALIZE, In := rtb_S_in, KL15_CM_Reset := rtb_S_in);
        DO_KL15_BB1 := i0_Chart_m.Out;
        (* Outport: '<Root>/DO_KL15_BB2' *)
        i1_Chart_m(ssMethodType := SS_INITIALIZE, In := rtb_S_in, KL15_CM_Reset := rtb_S_in);
        DO_KL15_BB2 := i1_Chart_m.Out;
        (* Outport: '<Root>/DO_KL15_BB3' *)
        i2_Chart_m(ssMethodType := SS_INITIALIZE, In := rtb_S_in, KL15_CM_Reset := rtb_S_in);
        DO_KL15_BB3 := i2_Chart_m.Out;
        i0_ChartBatt1(ssMethodType := SS_INITIALIZE, BattAvailable_LiBa := rtb_S_in, BattAvailable_Actia := rtb_IP_boBatt1_Actia_Availability);
        rtb_BattSelect_f := i0_ChartBatt1.BattSelect;
        i0_Chartbatt2(ssMethodType := SS_INITIALIZE, BattAvailable_LiBa := rtb_S_in, BattAvailable_Actia := rtb_IP_boBatt1_Actia_Availability);
        rtb_BattSelect := i0_Chartbatt2.BattSelect;
        i0_ChartBatt3(ssMethodType := SS_INITIALIZE, BattAvailable_LiBa := rtb_S_in, BattAvailable_Actia := rtb_IP_boBatt1_Actia_Availability);
        rtb_BattSelect_i := i0_ChartBatt3.BattSelect;
        (* SystemInitialize for Atomic SubSystem: '<Root>/ChiefMaster' *)
        (* SystemInitialize for Enabled SubSystem: '<S201>/Subsystem' *)
        (* SystemInitialize for DataTypeConversion: '<S209>/Data Type Conversion2' incorporates:
         *  Outport: '<S209>/Batt1_MyStatus1_Databus' *)
        IP_boBatt1_HV_REL_ON := FALSE;
        (* SystemInitialize for DataTypeConversion: '<S209>/Data Type Conversion5' incorporates:
         *  Outport: '<S209>/Batt1_MyStatus1_Databus' *)
        IP_boBatt1_SDERR_activ := FALSE;
        (* SystemInitialize for DataTypeConversion: '<S209>/Data Type Conversion6' incorporates:
         *  Outport: '<S209>/Batt1_MyStatus1_Databus' *)
        IP_boBatt1_ERROR_activ := FALSE;
        (* SystemInitialize for DataTypeConversion: '<S209>/Data Type Conversion7' incorporates:
         *  Outport: '<S209>/Batt1_MyStatus1_Databus' *)
        IP_boBatt1_WARNING_activ := FALSE;
        (* SystemInitialize for DataTypeConversion: '<S209>/Data Type Conversion8' incorporates:
         *  Outport: '<S209>/Batt1_MyStatus1_Databus' *)
        IP_boBatt1_Insulation_ready_and_OK := FALSE;
        (* End of SystemInitialize for SubSystem: '<S201>/Subsystem' *)
        (* End of SystemInitialize for SubSystem: '<Root>/ChiefMaster' *)
        i0_Lib_InputProcessing_state(ssMethodType := SS_INITIALIZE, Timeout := rtb_S_in, Data_In := rtb_ExtractDesiredBits_b13);
        DataTypeConversion_c := i0_Lib_InputProcessing_state.u8Data_Out;
        (* SystemInitialize for Atomic SubSystem: '<Root>/ChiefMaster' *)
        (* SystemInitialize for Enabled SubSystem: '<S262>/Subsystem' *)
        (* SystemInitialize for DataTypeConversion: '<S270>/Data Type Conversion2' incorporates:
         *  Outport: '<S270>/Batt2_MyStatus1_Databus' *)
        IP_boBatt2_HV_REL_ON := FALSE;
        (* SystemInitialize for DataTypeConversion: '<S270>/Data Type Conversion5' incorporates:
         *  Outport: '<S270>/Batt2_MyStatus1_Databus' *)
        IP_boBatt2_SDERR_activ := FALSE;
        (* SystemInitialize for DataTypeConversion: '<S270>/Data Type Conversion6' incorporates:
         *  Outport: '<S270>/Batt2_MyStatus1_Databus' *)
        IP_boBatt2_ERROR_activ := FALSE;
        (* SystemInitialize for DataTypeConversion: '<S270>/Data Type Conversion7' incorporates:
         *  Outport: '<S270>/Batt2_MyStatus1_Databus' *)
        IP_boBatt2_WARNING_activ := FALSE;
        (* SystemInitialize for DataTypeConversion: '<S270>/Data Type Conversion8' incorporates:
         *  Outport: '<S270>/Batt2_MyStatus1_Databus' *)
        IP_boBatt2_Insulation_ready_and_OK := FALSE;
        (* End of SystemInitialize for SubSystem: '<S262>/Subsystem' *)
        (* End of SystemInitialize for SubSystem: '<Root>/ChiefMaster' *)
        i1_Lib_InputProcessing_state(ssMethodType := SS_INITIALIZE, Timeout := rtb_S_in, Data_In := rtb_ExtractDesiredBits_b13);
        DataTypeConversion_i := i1_Lib_InputProcessing_state.u8Data_Out;
        (* SystemInitialize for Atomic SubSystem: '<Root>/ChiefMaster' *)
        (* SystemInitialize for Enabled SubSystem: '<S323>/Subsystem' *)
        (* SystemInitialize for DataTypeConversion: '<S331>/Data Type Conversion2' incorporates:
         *  Outport: '<S331>/Batt3_MyStatus1_Databus' *)
        IP_boBatt3_HV_REL_ON := FALSE;
        (* SystemInitialize for DataTypeConversion: '<S331>/Data Type Conversion5' incorporates:
         *  Outport: '<S331>/Batt3_MyStatus1_Databus' *)
        IP_boBatt3_SDERR_activ := FALSE;
        (* SystemInitialize for DataTypeConversion: '<S331>/Data Type Conversion6' incorporates:
         *  Outport: '<S331>/Batt3_MyStatus1_Databus' *)
        IP_boBatt3_ERROR_activ := FALSE;
        (* SystemInitialize for DataTypeConversion: '<S331>/Data Type Conversion7' incorporates:
         *  Outport: '<S331>/Batt3_MyStatus1_Databus' *)
        IP_boBatt3_WARNING_activ := FALSE;
        (* SystemInitialize for DataTypeConversion: '<S331>/Data Type Conversion8' incorporates:
         *  Outport: '<S331>/Batt3_MyStatus1_Databus' *)
        IP_boBatt3_Insulation_ready_and_OK := FALSE;
        (* End of SystemInitialize for SubSystem: '<S323>/Subsystem' *)
        (* End of SystemInitialize for SubSystem: '<Root>/ChiefMaster' *)
        i2_Lib_InputProcessing_state(ssMethodType := SS_INITIALIZE, Timeout := rtb_S_in, Data_In := rtb_ExtractDesiredBits_b13);
        DataTypeConversion := i2_Lib_InputProcessing_state.u8Data_Out;
        (* SystemInitialize for Atomic SubSystem: '<Root>/ChiefMaster' *)
        (* SystemInitialize for Enabled SubSystem: '<S203>/Subsystem' *)
        (* SystemInitialize for DataTypeConversion: '<S232>/Data Type Conversion2' incorporates:
         *  Outport: '<S232>/IP_boBatt1_HV_relay_PLUS_Sense' *)
        IP_boBatt1_HV_relay_PLUS_Sense := FALSE;
        (* SystemInitialize for DataTypeConversion: '<S232>/Data Type Conversion4' incorporates:
         *  Outport: '<S232>/IP_boBatt1_HV_relay_MINUS_Sense' *)
        IP_boBatt1_HV_relay_MINUS_Sense := FALSE;
        (* SystemInitialize for DataTypeConversion: '<S232>/Data Type Conversion5' incorporates:
         *  Outport: '<S232>/IP_boBatt1_IMD_active' *)
        IP_boBatt1_IMD_active := FALSE;
        (* End of SystemInitialize for SubSystem: '<S203>/Subsystem' *)
        

        (* SystemInitialize for Enabled SubSystem: '<S264>/Subsystem' *)
        (* SystemInitialize for DataTypeConversion: '<S293>/Data Type Conversion2' incorporates:
         *  Outport: '<S293>/IP_boBatt2_HV_relay_PLUS_Sense' *)
        IP_boBatt2_HV_relay_PLUS_Sense := FALSE;
        (* SystemInitialize for DataTypeConversion: '<S293>/Data Type Conversion4' incorporates:
         *  Outport: '<S293>/IP_boBatt2_HV_relay_MINUS_Sense' *)
        IP_boBatt2_HV_relay_MINUS_Sense := FALSE;
        (* SystemInitialize for DataTypeConversion: '<S293>/Data Type Conversion5' incorporates:
         *  Outport: '<S293>/IP_boBatt2_IMD_active' *)
        IP_boBatt2_IMD_active := FALSE;
        (* End of SystemInitialize for SubSystem: '<S264>/Subsystem' *)
        

        (* SystemInitialize for Enabled SubSystem: '<S325>/Subsystem' *)
        (* SystemInitialize for DataTypeConversion: '<S354>/Data Type Conversion2' incorporates:
         *  Outport: '<S354>/IP_boBatt3_HV_relay_PLUS_Sense' *)
        IP_boBatt3_HV_relay_PLUS_Sense := FALSE;
        (* SystemInitialize for DataTypeConversion: '<S354>/Data Type Conversion4' incorporates:
         *  Outport: '<S354>/IP_boBatt3_HV_relay_MINUS_Sense' *)
        IP_boBatt3_HV_relay_MINUS_Sense := FALSE;
        (* SystemInitialize for DataTypeConversion: '<S354>/Data Type Conversion5' incorporates:
         *  Outport: '<S354>/IP_boBatt3_IMD_active' *)
        IP_boBatt3_IMD_active := FALSE;
        (* End of SystemInitialize for SubSystem: '<S325>/Subsystem' *)
        (* End of SystemInitialize for SubSystem: '<Root>/ChiefMaster' *)
        

        (* Constant: '<S768>/Constant1' *)
        i2_IMD_OK(ssMethodType := SS_INITIALIZE, IP_boBMS_InsulationReadyOK := DI_IMD_FB_BB1, Req_IMD := rtb_IP_boBatt1_Actia_Availability, IT_u8IMD_DelayTime_s_g := IT_u8IMD_DelayTime_s);
        rtb_S_in := i2_IMD_OK.IMD_OK_i;
        (* Constant: '<S766>/Constant1' *)
        i0_IMD_OK(ssMethodType := SS_INITIALIZE, IP_boBMS_InsulationReadyOK := DI_IMD_FB_BB2, Req_IMD := rtb_Delay_dl, IT_u8IMD_DelayTime_s_g := IT_u8IMD_DelayTime_s);
        rtb_IP_boBatt1_Actia_Availability := i0_IMD_OK.IMD_OK_i;
        (* Constant: '<S767>/Constant1' *)
        i1_IMD_OK(ssMethodType := SS_INITIALIZE, IP_boBMS_InsulationReadyOK := DI_IMD_FB_BB3, Req_IMD := rtb_Delay_j, IT_u8IMD_DelayTime_s_g := IT_u8IMD_DelayTime_s);
        rtb_Delay_dl := i1_IMD_OK.IMD_OK_i;
        i0_IMDOK_Input_Delay(ssMethodType := SS_INITIALIZE, In := rtb_Delay_j);
        rtb_out_l := i0_IMDOK_Input_Delay.out;
        i1_IMDOK_Input_Delay(ssMethodType := SS_INITIALIZE, In := rtb_Delay_j);
        rtb_out_l := i1_IMDOK_Input_Delay.out;
        i2_IMDOK_Input_Delay(ssMethodType := SS_INITIALIZE, In := rtb_Delay_j);
        rtb_out_l := i2_IMDOK_Input_Delay.out;
        i0_REQ_HV_ON_Batt(ssMethodType := SS_INITIALIZE, IsolationMeasurementRequest := rtb_IT_boUDC_EV_IsolationMeasurementRequest, IP_boChargeStop_Pressed := rtb_IT_boChargeStop_Button, SafeToSD_BB1 := rtb_Delay_j, SafeToSD_BB2 := rtb_Delay_j, SafeToSD_BB3 := rtb_FL_boCMSleep, KL15_CM_disable := rtb_FL_boKL15_Disable, SDError_BB1 := rtb_IT_boBMS_SDError_BB1, SDError_BB2 := rtb_IT_boBMS_SDError_BB1, SDError_BB3 := rtb_IT_boBMS_SDError_BB1, InsulationReadyOK_B1 := rtb_IT_boBMS_SDError_BB1, InsulationReadyOK_B2 := rtb_IT_boBMS_SDError_BB1, InsulationReadyOK_B3 := rtb_IT_boBMS_SDError_BB1, IMD_Active_BB1 := rtb_IT_boBMS_SDError_BB1, IMD_Active_BB2 := rtb_IT_boBMS_SDError_BB1, IMD_Active_BB3 := rtb_IT_boBMS_SDError_BB1, Software_Reset_KL15_BB3 := DINT_TO_LREAL(rtb_UnitDelay5), Software_Reset_KL15_BB2 := DINT_TO_LREAL(rtb_UnitDelay5), Software_Reset_KL15_BB1 := DINT_TO_LREAL(rtb_UnitDelay5), FL_boSafeToCloseHV_BB1 := rtb_Delay_j, FL_boSafeToCloseHV_BB2 := rtb_FL_boSS_HVIL_NOK, FL_boSafeToCloseHV_BB3 := rtb_FL_boHVC_AllCellBalanced, FL_boST_REQ_HV_Open_BB1 := rtb_Delay_j, FL_boST_REQ_HV_Open_BB2 := rtb_Delay_j, FL_boST_REQ_HV_Open_BB3 := rtb_Delay_j, FL_boSystem_SD := rtb_Delay_j, HV_Minus_Sense_BB1 := rtb_Delay_j, HV_Plus_Sense_BB1 := rtb_Delay_j, HV_Minus_Sense_BB2 := rtb_Delay_j, HV_Plus_Sense_BB2 := rtb_Delay_j, HV_Minus_Sense_BB3 := rtb_Delay_j, HV_Plus_Sense_BB3 := rtb_Delay_j, HV_REL_ON_BB2 := rtb_IT_boBMS_SDError_BB1, HV_REL_ON_BB1 := rtb_IT_boBMS_SDError_BB1, HV_REL_ON_BB3 := rtb_IT_boBMS_SDError_BB1, FL_boMainHV_SD_OK := rtb_Delay_j, FL_boMainHV_PlusMinus_Status := rtb_Delay_j);
        ContactorState_i := i0_REQ_HV_ON_Batt.FL_u8ContactorState_BB1;
        ContactorState_f := i0_REQ_HV_ON_Batt.FL_u8ContactorState_BB2;
        ContactorState := i0_REQ_HV_ON_Batt.FL_u8ContactorState_BB3;
        REQ_HV_ON_a := i0_REQ_HV_ON_Batt.FL_boREQ_HV_ON_BB1;
        REQ_HV_ON_d := i0_REQ_HV_ON_Batt.FL_boREQ_HV_ON_BB2;
        REQ_HV_ON := i0_REQ_HV_ON_Batt.FL_boREQ_HV_ON_BB3;
        rtb_Contactor_FB_State_h := i0_REQ_HV_ON_Batt.FL_u8Contactor_FB_State_BB1;
        rtb_Contactor_FB_State_g := i0_REQ_HV_ON_Batt.FL_u8Contactor_FB_State_BB2;
        rtb_Contactor_FB_State := i0_REQ_HV_ON_Batt.FL_u8Contactor_FB_State_BB3;
        (* SystemInitialize for Atomic SubSystem: '<Root>/ChiefMaster' *)
        (* SystemInitialize for Chart: '<S13>/Chart_REQ_MAIN_Precharge' *)
        is_active_c19_ChiefMaster := 0;
        is_c19_ChiefMaster := ChiefMaster_IN_NO_ACTIVE_CHILD_f;
        i0_Chart_PrechargeStatus(ssMethodType := SS_INITIALIZE, REQ_MainHV_ON_Precharge := FALSE, LoadCurrent := rtb_Delay_j, LoadVoltage := DINT_TO_REAL(rtb_Add_kr), SystemVoltage := rtb_Min, KL15_CM_diable := rtb_FL_boKL15_Disable, MainHV_Minus_Status := DINT_TO_LREAL(rtb_UnitDelay5));
        Precharge_Satus := i0_Chart_PrechargeStatus.Precharge_Satus;
        (* SystemInitialize for Chart: '<S13>/delay' *)
        temporalCounter_i1_m(timerAction := 1, maxTime := 0);
        is_active_c4_ChiefMaster := 0;
        is_c4_ChiefMaster := ChiefMaster_IN_NO_ACTIVE_CHILD_f;
        (* End of SystemInitialize for SubSystem: '<Root>/ChiefMaster' *)
        

        (* Constant: '<S388>/Constant4' incorporates:
         *  Constant: '<S388>/Constant'
         *  Constant: '<S388>/Constant1'
         *  Constant: '<S388>/Constant2'
         *  Constant: '<S388>/Constant3' *)
        i0_Chart_Hysteresis_LowActive(ssMethodType := SS_INITIALIZE, sSignal := AI_MainHV_Minus_FB, boInitial_Value := FALSE, boValue_Activated := TRUE, boValue_Deactivated := FALSE, sLB := 5000.0, b_sUB := 10000.0);
        boOutput_n := i0_Chart_Hysteresis_LowActive.boOutput;
        (* Constant: '<S382>/Constant4' incorporates:
         *  Constant: '<S382>/Constant'
         *  Constant: '<S382>/Constant1'
         *  Constant: '<S382>/Constant2'
         *  Constant: '<S382>/Constant3' *)
        i0_Chart_Hysteresis_HighActive(ssMethodType := SS_INITIALIZE, sSignal := AI_EmergencyButton_NC, boInitial_Value := FALSE, boValue_Activated := TRUE, boValue_Deactivated := FALSE, sLB := 2000.0, b_sUB := 8000.0);
        boOutput_h := i0_Chart_Hysteresis_HighActive.boOutput;
        (* Constant: '<S383>/Constant4' incorporates:
         *  Constant: '<S383>/Constant'
         *  Constant: '<S383>/Constant1'
         *  Constant: '<S383>/Constant2'
         *  Constant: '<S383>/Constant3' *)
        i1_Chart_Hysteresis_HighActive(ssMethodType := SS_INITIALIZE, sSignal := AI_EmergencyButton_NO, boInitial_Value := FALSE, boValue_Activated := TRUE, boValue_Deactivated := FALSE, sLB := 18000.0, b_sUB := 22000.0);
        boOutput_k := i1_Chart_Hysteresis_HighActive.boOutput;
        (* Constant: '<S384>/Constant4' incorporates:
         *  Constant: '<S384>/Constant'
         *  Constant: '<S384>/Constant1'
         *  Constant: '<S384>/Constant2'
         *  Constant: '<S384>/Constant3' *)
        i2_Chart_Hysteresis_HighActive(ssMethodType := SS_INITIALIZE, sSignal := AI_HVIL_BDU, boInitial_Value := FALSE, boValue_Activated := TRUE, boValue_Deactivated := FALSE, sLB := 12000.0, b_sUB := 15000.0);
        boOutput_l := i2_Chart_Hysteresis_HighActive.boOutput;
        (* Constant: '<S384>/Constant5' *)
        i0_HVIL_Input_Delay(ssMethodType := SS_INITIALIZE, HVIL_IN := boOutput_l, IP_HVIL_Delay_ms := IP_u8HVIL_Delay_ms);
        rtb_out_l := i0_HVIL_Input_Delay.out;
        (* Constant: '<S385>/Constant4' incorporates:
         *  Constant: '<S385>/Constant'
         *  Constant: '<S385>/Constant1'
         *  Constant: '<S385>/Constant2'
         *  Constant: '<S385>/Constant3' *)
        i3_Chart_Hysteresis_HighActive(ssMethodType := SS_INITIALIZE, sSignal := AI_HVIL_Component, boInitial_Value := FALSE, boValue_Activated := TRUE, boValue_Deactivated := FALSE, sLB := 12000.0, b_sUB := 15000.0);
        boOutput_p := i3_Chart_Hysteresis_HighActive.boOutput;
        (* Constant: '<S385>/Constant5' *)
        i1_HVIL_Input_Delay(ssMethodType := SS_INITIALIZE, HVIL_IN := boOutput_p, IP_HVIL_Delay_ms := IP_u8HVIL_Delay_ms);
        rtb_FL_boHVC_AllCellBalanced := i1_HVIL_Input_Delay.out;
        (* Constant: '<S386>/Constant4' incorporates:
         *  Constant: '<S386>/Constant'
         *  Constant: '<S386>/Constant1'
         *  Constant: '<S386>/Constant2'
         *  Constant: '<S386>/Constant3' *)
        i4_Chart_Hysteresis_HighActive(ssMethodType := SS_INITIALIZE, sSignal := AI_HVIL_Battery, boInitial_Value := FALSE, boValue_Activated := TRUE, boValue_Deactivated := FALSE, sLB := 12000.0, b_sUB := 15000.0);
        boOutput_f := i4_Chart_Hysteresis_HighActive.boOutput;
        (* Constant: '<S386>/Constant5' *)
        i2_HVIL_Input_Delay(ssMethodType := SS_INITIALIZE, HVIL_IN := boOutput_f, IP_HVIL_Delay_ms := IP_u8HVIL_Delay_ms);
        rtb_out_n := i2_HVIL_Input_Delay.out;
        i3_Chart_SetDominantSwitch(ssMethodType := SS_INITIALIZE, boData_In := rtb_Delay_j, boReset := rtb_FL_boKL15_Reset);
        rtb_boData_Out := i3_Chart_SetDominantSwitch.boData_Out;
        i0_EmergencySD(ssMethodType := SS_INITIALIZE, FL_boKL15_Reset := rtb_FL_boKL15_Reset, IT_boEmergencySwitch_NC := rtb_IT_sHW_EmergencyButton_NC, IT_boEmergencySwitch_NO := rtb_IT_boHW_EmergencyButton_NO, IT_boHW_HVIL_BDU := rtb_IT_boHW_HVIL_BDU, IT_boHW_HVIL_Components := rtb_IT_boHW_HVIL_BDU, IT_boHW_HVIL_Battery := rtb_IT_boHW_HVIL_BDU, IT_boHW_HVIL_Overrule := rtb_IT_boHW_HVIL_BDU, IT_boHW_ResetButton_LED_NO_State := rtb_boData_Out);
        rtb_Delay_j := i0_EmergencySD.FL_boSS_System_ESD;
        rtb_Out := i0_EmergencySD.FL_u8SS_EmergencyStopState;
        rtb_FL_boSS_HVIL_NOK := i0_EmergencySD.FL_boHVIL_NOK;
        i0_Input_Delay(ssMethodType := SS_INITIALIZE, IP_u8HW_IN_delay_ms_m := b_Constant, Input := DI_Proximity_BB1);
        rtb_IT_boHW_HVIL_BDU := i0_Input_Delay.out;
        i1_Input_Delay(ssMethodType := SS_INITIALIZE, IP_u8HW_IN_delay_ms_m := Constant_n, Input := DI_Proximity_BB2);
        rtb_out_i := i1_Input_Delay.out;
        i2_Input_Delay(ssMethodType := SS_INITIALIZE, IP_u8HW_IN_delay_ms_m := Constant_o, Input := DI_Proximity_BB3);
        rtb_out_ne := i2_Input_Delay.out;
        i0_SDError(ssMethodType := SS_INITIALIZE, FL_boKL15_Reset := rtb_FL_boKL15_Reset, IT_Databus := rtb_ExtractDesiredBits_b13, IT_Databus_m := rtb_IT_boBMS_SDError_BB1, IT_Databus_n := rtb_IT_boBMS_SDError_BB1, IT_Databus_a := rtb_IT_boBMS_SDError_BB1, IT_Databus_o := rtb_IT_boBMS_SDError_BB1, IT_Databus_or := rtb_IT_boBMS_SDError_BB1, IT_Databus_i := rtb_IT_boBMS_SDError_BB1, IT_Databus_c := rtb_Min, IT_Databus_o3 := rtb_Min, IT_Databus_e := rtb_Min, IT_Databus_n0 := rtb_IT_boChargeStop_Button, IT_Databus_ep := rtb_IT_boChargeStop_Button, IT_Databus_l := rtb_IT_boChargeStop_Button, IT_Databus_f := rtb_IT_boBMS_SDError_BB1, IT_Databus_k := rtb_IT_boBMS_SDError_BB1, IT_Databus_g := rtb_IT_boBMS_SDError_BB1, IT_Databus_b := rtb_IT_boBMS_SDError_BB1, IT_Databus_d := rtb_AND_l2, IT_Databus_h := rtb_IT_boBMS_SDError_BB1, IT_Databus_j := rtb_AND_ni, IT_Databus_ja := rtb_IT_boBMS_SDError_BB1, IT_Databus_if := rtb_AND_ma, FL_BDUControl_Databus := MainHV_Minus_Status, FL_BDUControl_Databus_o := MainHV_Plus_Status, FL_BDUControl_Databus_n := Precharge_Satus, FL_BatteryBox_HVControl_Databus := REQ_HV_ON_a, FL_BatteryBox_HVControl_Databus_b := REQ_HV_ON_d, FL_BatteryBox_HVControl_Databus_a := REQ_HV_ON, FL_u8SS_EmergencySD := rtb_Delay_j);
        System_Error := i0_SDError.FL_boSS_System_SD;
        rtb_System_SD_ErrorCode := i0_SDError.FL_u8SS_System_SD_ErrorCode;
        (* Constant: '<S110>/Constant5' incorporates:
         *  Constant: '<S110>/Constant6' *)
        i0_BattChargeFcn(ssMethodType := SS_INITIALIZE, MaxChargeCurr_fb := rtb_UnitDelay, MaxChargeCurrentBatt := rtb_Min, ChargeStopPressed := rtb_IT_boChargeStop_Button, HV_ON_Batt1 := rtb_IT_boBMS_SDError_BB1, HV_ON_Batt2 := rtb_IT_boBMS_SDError_BB1, HV_ON_Batt3 := rtb_IT_boBMS_SDError_BB1, Ibatt1 := rtb_Min, Ibatt2 := rtb_Min, Ibatt3 := rtb_Min, Fcn_available := rtb_IT_boChargeStop_Button, CurrentReductionConstant := rtb_Switch3, CurrentLB_f := CurrentLB, CurrentUB_c := CurrentUB);
        FL_sST_MaxChargeCurrent := i0_BattChargeFcn.FL_sST_MaxChargeCurrent;
        REQ_HV_Open_Batt2 := i0_BattChargeFcn.REQ_HV_Open_Batt2;
        REQ_HV_Open_Batt3 := i0_BattChargeFcn.REQ_HV_Open_Batt3;
        REQ_HV_Open_Batt1 := i0_BattChargeFcn.REQ_HV_Open_Batt1;
        BatteryReadyToShutDown := i0_BattChargeFcn.BatteryReadyToShutDown;
        (* SystemInitialize for Atomic SubSystem: '<Root>/ChiefMaster' *)
        (* SystemInitialize for Chart: '<S13>/delay' *)
        i0_Chart_REQ_MAIN_MINUS(ssMethodType := SS_INITIALIZE, In := FALSE, CM_SafeToSD := rtb_IT_boChargeStop_Button, KL15_CM_disable := rtb_FL_boKL15_Disable, System_ESD := rtb_IT_boChargeStop_Button, System_SD := rtb_UnitDelay1_d, b_Reset := rtb_FL_boSS_BDU_Reset);
        REQ_MainHV_ON_MINUS_g := i0_Chart_REQ_MAIN_MINUS.REQ_MainHV_ON_MINUS;
        (* End of SystemInitialize for SubSystem: '<Root>/ChiefMaster' *)
        i0_Chart_WeldingDetection(ssMethodType := SS_INITIALIZE, LoadVtg := DINT_TO_REAL(rtb_Add_kr), SystemVtg := rtb_Min, In := rtb_IT_boChargeStop_Button);
        MainHV_Minus_Welded := i0_Chart_WeldingDetection.MainHV_Minus_Welded;
        MainHV_Plus_Welded := i0_Chart_WeldingDetection.MainHV_Plus_Welded;
        REQ_MainHV_ON_MINUS := i0_Chart_WeldingDetection.REQ_MainHV_ON_MINUS;
        REQ_MainHV_ON_PLUS := i0_Chart_WeldingDetection.REQ_MainHV_ON_PLUS;
        WeldingDetection_Status := i0_Chart_WeldingDetection.WeldingDetection_Status;
        (* SystemInitialize for Atomic SubSystem: '<Root>/ChiefMaster' *)
        (* SystemInitialize for Chart: '<S21>/Chart4' *)
        is_active_c46_ChiefMaster := 0;
        is_c46_ChiefMaster := ChiefMaster_IN_NO_ACTIVE_CHILD_f;
        (* SystemInitialize for Chart: '<S20>/Chart_Main_Minus_Status' *)
        temporalCounter_i1_k(timerAction := 1, maxTime := 0);
        is_active_c40_ChiefMaster := 0;
        is_c40_ChiefMaster := ChiefMaster_IN_NO_ACTIVE_CHILD_f;
        MainHV_Minus_Status := 0.0;
        (* End of SystemInitialize for SubSystem: '<Root>/ChiefMaster' *)
        

        (* Constant: '<S390>/Constant4' incorporates:
         *  Constant: '<S390>/Constant'
         *  Constant: '<S390>/Constant1'
         *  Constant: '<S390>/Constant2'
         *  Constant: '<S390>/Constant3' *)
        i2_Chart_Hysteresis_LowActive(ssMethodType := SS_INITIALIZE, sSignal := AI_MainHV_Plus_FB, boInitial_Value := FALSE, boValue_Activated := TRUE, boValue_Deactivated := FALSE, sLB := 5000.0, b_sUB := 10000.0);
        boOutput_o := i2_Chart_Hysteresis_LowActive.boOutput;
        (* SystemInitialize for Atomic SubSystem: '<Root>/ChiefMaster' *)
        (* SystemInitialize for Chart: '<S20>/Chart_Main_Plus_Status' *)
        temporalCounter_i1_he(timerAction := 1, maxTime := 0);
        is_active_c41_ChiefMaster := 0;
        is_c41_ChiefMaster := ChiefMaster_IN_NO_ACTIVE_CHILD_f;
        MainHV_Plus_Status := 0.0;
        (* End of SystemInitialize for SubSystem: '<Root>/ChiefMaster' *)
        

        (* Constant: '<S389>/Constant4' incorporates:
         *  Constant: '<S389>/Constant'
         *  Constant: '<S389>/Constant1'
         *  Constant: '<S389>/Constant2'
         *  Constant: '<S389>/Constant3' *)
        i1_Chart_Hysteresis_LowActive(ssMethodType := SS_INITIALIZE, sSignal := AI_DCHV_Minus_FB, boInitial_Value := FALSE, boValue_Activated := TRUE, boValue_Deactivated := FALSE, sLB := 5000.0, b_sUB := 10000.0);
        boOutput_a := i1_Chart_Hysteresis_LowActive.boOutput;
        (* SystemInitialize for Atomic SubSystem: '<Root>/ChiefMaster' *)
        (* SystemInitialize for Chart: '<S23>/Chart_DCMinus_Status' *)
        temporalCounter_i1_n(timerAction := 1, maxTime := 0);
        is_active_c53_ChiefMaster := 0;
        is_c53_ChiefMaster := ChiefMaster_IN_NO_ACTIVE_CHILD_f;
        (* End of SystemInitialize for SubSystem: '<Root>/ChiefMaster' *)
        

